C03636=1030.587,97.043,400.523,168.711,44.180,158.272
C03637=1030.581,96.794,400.543,168.708,44.181,158.272
C03638=1030.575,96.545,400.561,168.706,44.183,158.272
C03639=1030.569,96.295,400.580,168.703,44.185,158.272
C03640=1030.563,96.046,400.599,168.701,44.187,158.272
C03641=1030.556,95.797,400.618,168.699,44.189,158.273
C03642=1030.551,95.548,400.637,168.696,44.191,158.273
C03643=1030.544,95.298,400.656,168.694,44.193,158.273
C03644=1030.539,95.049,400.675,168.691,44.195,158.273
C03645=1030.532,94.800,400.694,168.689,44.197,158.273
C03646=1030.526,94.550,400.713,168.687,44.198,158.273
C03647=1030.520,94.301,400.731,168.684,44.200,158.273
C03648=1030.514,94.053,400.751,168.682,44.202,158.274
C03649=1030.508,93.803,400.770,168.679,44.204,158.274
C03650=1030.501,93.554,400.789,168.677,44.206,158.274
C03651=1030.496,93.305,400.808,168.675,44.208,158.274
C03652=1030.489,93.056,400.827,168.673,44.210,158.274
C03653=1030.483,92.806,400.846,168.670,44.211,158.274
C03654=1030.476,92.521,400.866,168.667,44.213,158.274
C03655=1030.469,92.236,400.888,168.665,44.215,158.275
C03656=1030.462,91.950,400.911,168.661,44.217,158.275
C03657=1030.455,91.665,400.932,168.659,44.219,158.275
C03658=1030.449,91.416,400.951,168.656,44.221,158.275
C03659=1030.443,91.166,400.970,168.654,44.223,158.275
C03660=1030.437,90.918,400.988,168.652,44.225,158.275
C03661=1030.431,90.669,401.007,168.649,44.227,158.275
C03662=1030.425,90.419,401.026,168.647,44.229,158.275
C03663=1030.419,90.170,401.045,168.644,44.231,158.276
C03664=1030.413,89.921,401.064,168.642,44.232,158.276
C03665=1030.407,89.672,401.083,168.640,44.234,158.276
C03666=1030.400,89.422,401.101,168.637,44.236,158.276
C03667=1030.394,89.173,401.119,168.635,44.238,158.276
C03668=1030.388,88.923,401.138,168.632,44.240,158.276
C03669=1030.382,88.674,401.157,168.631,44.242,158.277
C03670=1030.376,88.425,401.176,168.628,44.244,158.277
C03671=1030.369,88.176,401.194,168.625,44.245,158.277
C03672=1030.363,87.926,401.212,168.623,44.247,158.277
C03673=1030.357,87.677,401.231,168.620,44.249,158.277
C03674=1030.351,87.429,401.249,168.618,44.252,158.277
C03675=1030.345,87.179,401.269,168.616,44.254,158.278
C03676=1030.339,86.929,401.286,168.614,44.256,158.278
C03677=1030.333,86.680,401.305,168.611,44.257,158.278
C03678=1030.326,86.431,401.324,168.608,44.259,158.278
C03679=1030.320,86.182,401.342,168.606,44.261,158.278
C03680=1030.314,85.932,401.360,168.604,44.263,158.278
C03681=1030.307,85.683,401.379,168.602,44.265,158.278
C03682=1030.301,85.434,401.398,168.599,44.267,158.279
C03683=1030.296,85.185,401.417,168.597,44.269,158.279
C03684=1030.290,84.936,401.434,168.594,44.271,158.279
C03685=1030.283,84.686,401.453,168.591,44.273,158.279
C03686=1030.277,84.437,401.472,168.590,44.274,158.279
C03687=1030.271,84.188,401.490,168.587,44.276,158.279
C03688=1030.264,83.938,401.508,168.585,44.278,158.279
C03689=1030.258,83.689,401.527,168.582,44.280,158.280
C03690=1030.252,83.441,401.545,168.579,44.282,158.280
C03691=1030.246,83.191,401.563,168.578,44.284,158.280
C03692=1030.240,82.942,401.582,168.575,44.286,158.280
C03693=1030.234,82.693,401.601,168.573,44.288,158.280
C03694=1030.228,82.443,401.619,168.570,44.290,158.280
C03695=1030.222,82.194,401.637,168.567,44.291,158.280
C03696=1030.216,81.945,401.655,168.566,44.293,158.281
C03697=1030.209,81.696,401.674,168.563,44.295,158.281
C03698=1030.203,81.446,401.693,168.561,44.297,158.281
C03699=1030.197,81.197,401.710,168.558,44.299,158.281
C03700=1030.191,80.948,401.729,168.557,44.301,158.281
C03701=1030.185,80.698,401.747,168.554,44.303,158.281
C03702=1030.179,80.449,401.766,168.551,44.304,158.281
C03703=1030.173,80.200,401.785,168.549,44.306,158.282
C03704=1030.166,79.950,401.803,168.546,44.308,158.282
C03705=1030.161,79.702,401.821,168.545,44.310,158.282
C03706=1030.155,79.452,401.839,168.542,44.312,158.282
C03707=1030.148,79.203,401.857,168.539,44.314,158.282
C03708=1030.142,78.953,401.875,168.537,44.316,158.282
C03709=1030.136,78.705,401.894,168.535,44.318,158.282
C03710=1030.130,78.456,401.912,168.533,44.319,158.283
C03711=1030.124,78.206,401.930,168.530,44.321,158.283
C03712=1030.118,77.957,401.949,168.528,44.323,158.283
C03713=1030.112,77.708,401.967,168.525,44.325,158.283
C03714=1030.106,77.458,401.984,168.523,44.327,158.283
C03715=1030.099,77.209,402.003,168.521,44.329,158.283
C03716=1030.093,76.959,402.021,168.518,44.331,158.283
C03717=1030.087,76.711,402.039,168.516,44.333,158.284
C03718=1030.080,76.425,402.060,168.513,44.335,158.284
C03719=1030.073,76.140,402.081,168.511,44.337,158.284
C03720=1030.066,75.855,402.102,168.508,44.339,158.284
C03721=1030.059,75.569,402.122,168.505,44.342,158.284
C03722=1030.053,75.320,402.140,168.503,44.344,158.284
C03723=1030.046,75.070,402.158,168.501,44.346,158.285
C03724=1030.040,74.821,402.175,168.498,44.348,158.285
C03725=1030.034,74.572,402.194,168.495,44.349,158.285
C03726=1030.028,74.322,402.212,168.493,44.351,158.285
C03727=1030.022,74.073,402.229,168.490,44.353,158.285
C03728=1030.016,73.824,402.248,168.489,44.355,158.285
C03729=1030.009,73.575,402.265,168.486,44.357,158.285
C03730=1030.003,73.325,402.283,168.483,44.359,158.286
C03731=1029.997,73.076,402.302,168.481,44.361,158.286
C03732=1029.991,72.827,402.320,168.478,44.363,158.286
C03733=1029.985,72.577,402.338,168.477,44.365,158.286
C03734=1029.978,72.329,402.355,168.474,44.366,158.286
C03735=1029.972,72.079,402.373,168.471,44.368,158.286
C03736=1029.966,71.829,402.391,168.469,44.370,158.286
C03737=1029.960,71.580,402.409,168.466,44.372,158.287
C03738=1029.954,71.331,402.427,168.465,44.374,158.287
C03739=1029.947,71.082,402.445,168.462,44.376,158.287
C03740=1029.942,70.833,402.462,168.460,44.378,158.287
C03741=1029.936,70.583,402.480,168.457,44.380,158.287
C03742=1029.929,70.334,402.499,168.456,44.382,158.287
C03743=1029.924,70.085,402.516,168.453,44.384,158.288
C03744=1029.917,69.835,402.534,168.450,44.386,158.288
C03745=1029.911,69.586,402.552,168.448,44.388,158.288
C03746=1029.905,69.337,402.569,168.445,44.390,158.288
C03747=1029.899,69.087,402.588,168.444,44.392,158.288
C03748=1029.892,68.838,402.605,168.441,44.394,158.288
C03749=1029.886,68.589,402.623,168.439,44.395,158.288
C03750=1029.880,68.339,402.641,168.436,44.397,158.289
C03751=1029.874,68.091,402.658,168.433,44.399,158.289
C03752=1029.868,67.841,402.676,168.432,44.401,158.289
C03753=1029.862,67.591,402.694,168.429,44.403,158.289
C03754=1029.855,67.343,402.711,168.427,44.405,158.289
C03755=1029.849,67.093,402.729,168.424,44.407,158.289
C03756=1029.842,66.844,402.746,168.421,44.409,158.289
C03757=1029.837,66.595,402.764,168.419,44.411,158.290
C03758=1029.831,66.345,402.782,168.418,44.413,158.290
C03759=1029.824,66.096,402.799,168.415,44.415,158.290
C03760=1029.818,65.847,402.817,168.412,44.417,158.290
C03761=1029.811,65.597,402.834,168.410,44.419,158.290
C03762=1029.806,65.348,402.852,168.407,44.421,158.290
C03763=1029.800,65.098,402.870,168.406,44.423,158.290
C03764=1029.793,64.850,402.887,168.403,44.424,158.291
C03765=1029.787,64.600,402.905,168.400,44.426,158.291
C03766=1029.781,64.351,402.922,168.398,44.428,158.291
C03767=1029.775,64.101,402.940,168.395,44.430,158.291
C03768=1029.768,63.852,402.957,168.394,44.432,158.291
C03769=1029.763,63.603,402.974,168.391,44.434,158.291
C03770=1029.756,63.353,402.992,168.389,44.437,158.292
C03771=1029.750,63.104,403.009,168.386,44.439,158.292
C03772=1029.743,62.855,403.027,168.384,44.440,158.292
C03773=1029.736,62.606,403.044,168.381,44.442,158.292
C03774=1029.731,62.356,403.061,168.379,44.445,158.292
C03775=1029.724,62.106,403.078,168.377,44.447,158.292
C03776=1029.718,61.858,403.095,168.374,44.449,158.293
C03777=1029.712,61.608,403.113,168.372,44.451,158.293
C03778=1029.706,61.359,403.130,168.369,44.453,158.293
C03779=1029.699,61.110,403.147,168.367,44.455,158.293
C03780=1029.692,60.860,403.164,168.364,44.457,158.293
C03781=1029.687,60.611,403.182,168.362,44.459,158.293
C03782=1029.679,60.325,403.201,168.359,44.462,158.294
C03783=1029.672,60.040,403.222,168.357,44.464,158.294
C03784=1029.665,59.755,403.241,168.354,44.466,158.294
C03785=1029.658,59.469,403.261,168.351,44.468,158.294
C03786=1029.651,59.220,403.278,168.348,44.470,158.294
C03787=1029.645,58.970,403.294,168.347,44.472,158.294
C03788=1029.639,58.720,403.312,168.344,44.475,158.295
C03789=1029.633,58.472,403.329,168.342,44.477,158.295
C03790=1029.626,58.222,403.346,168.339,44.478,158.295
C03791=1029.620,57.973,403.363,168.337,44.480,158.295
C03792=1029.614,57.723,403.381,168.334,44.482,158.295
C03793=1029.607,57.475,403.398,168.332,44.484,158.295
C03794=1029.601,57.225,403.415,168.330,44.487,158.296
C03795=1029.595,56.975,403.432,168.328,44.489,158.296
C03796=1029.588,56.726,403.449,168.325,44.491,158.296
C03797=1029.582,56.477,403.466,168.322,44.492,158.296
C03798=1029.576,56.227,403.483,168.320,44.494,158.296
C03799=1029.570,55.978,403.500,168.318,44.496,158.296
C03800=1029.563,55.729,403.518,168.316,44.498,158.296
C03801=1029.557,55.479,403.534,168.313,44.501,158.297
C03802=1029.550,55.230,403.551,168.311,44.503,158.297
C03803=1029.545,54.981,403.569,168.308,44.505,158.297
C03804=1029.538,54.731,403.585,168.305,44.507,158.297
C03805=1029.532,54.482,403.602,168.303,44.508,158.297
C03806=1029.526,54.233,403.619,168.301,44.510,158.297
C03807=1029.520,53.983,403.637,168.299,44.512,158.297
C03808=1029.514,53.734,403.654,168.296,44.514,158.298
C03809=1029.507,53.485,403.671,168.294,44.517,158.298
C03810=1029.502,53.235,403.688,168.291,44.519,158.298
C03811=1029.495,52.986,403.705,168.290,44.520,158.298
C03812=1029.489,52.736,403.721,168.287,44.522,158.298
C03813=1029.483,52.488,403.738,168.284,44.524,158.298
C03814=1029.477,52.238,403.756,168.282,44.526,158.299
C03815=1029.471,51.989,403.772,168.279,44.528,158.299
C03816=1029.464,51.739,403.790,168.277,44.530,158.299
C03817=1029.458,51.490,403.806,168.275,44.532,158.299
C03818=1029.452,51.241,403.823,168.273,44.534,158.299
C03819=1029.446,50.991,403.840,168.270,44.536,158.299
C03820=1029.439,50.742,403.857,168.268,44.538,158.300
C03821=1029.433,50.493,403.873,168.265,44.540,158.300
C03822=1029.427,50.243,403.891,168.262,44.542,158.300
C03823=1029.421,49.994,403.908,168.261,44.544,158.300
C03824=1029.415,49.744,403.925,168.258,44.546,158.300
C03825=1029.408,49.495,403.942,168.256,44.548,158.300
C03826=1029.402,49.246,403.958,168.253,44.550,158.300
C03827=1029.396,48.996,403.976,168.251,44.552,158.300
C03828=1029.390,48.747,403.992,168.249,44.554,158.301
C03829=1029.384,48.498,404.009,168.246,44.555,158.301
C03830=1029.377,48.248,404.026,168.244,44.557,158.301
C03831=1029.372,47.999,404.043,168.241,44.559,158.301
C03832=1029.366,47.750,404.060,168.239,44.561,158.301
C03833=1029.360,47.500,404.076,168.237,44.563,158.301
C03834=1029.353,47.251,404.093,168.235,44.565,158.301
C03835=1029.347,47.002,404.110,168.232,44.567,158.302
C03836=1029.342,46.753,404.127,168.229,44.569,158.302
C03837=1029.335,46.503,404.144,168.227,44.571,158.302
C03838=1029.329,46.254,404.161,168.225,44.573,158.302
C03839=1029.323,46.005,404.177,168.223,44.575,158.302
C03840=1029.317,45.754,404.194,168.220,44.576,158.302
C03841=1029.311,45.505,404.211,168.217,44.578,158.302
C03842=1029.305,45.256,404.228,168.215,44.580,158.302
C03843=1029.299,45.007,404.245,168.213,44.582,158.303
C03844=1029.292,44.757,404.261,168.211,44.584,158.303
C03845=1029.287,44.508,404.278,168.208,44.586,158.303
C03846=1029.279,44.222,404.297,168.206,44.588,158.303
C03847=1029.273,43.936,404.316,168.203,44.591,158.303
C03848=1029.265,43.651,404.336,168.200,44.593,158.303
C03849=1029.259,43.365,404.354,168.197,44.595,158.303
C03850=1029.253,43.115,404.372,168.194,44.597,158.304
C03851=1029.247,42.866,404.388,168.193,44.598,158.304
C03852=1029.241,42.617,404.404,168.190,44.600,158.304
C03853=1029.235,42.367,404.421,168.188,44.602,158.304
C03854=1029.228,42.118,404.438,168.185,44.604,158.304
C03855=1029.222,41.868,404.454,168.183,44.606,158.304
C03856=1029.216,41.619,404.470,168.180,44.609,158.304
C03857=1029.210,41.370,404.487,168.178,44.611,158.305
C03858=1029.203,41.120,404.503,168.176,44.613,158.305
C03859=1029.197,40.871,404.520,168.173,44.614,158.305
C03860=1029.191,40.622,404.537,168.171,44.616,158.305
C03861=1029.185,40.372,404.553,168.168,44.618,158.305
C03862=1029.179,40.122,404.569,168.166,44.620,158.305
C03863=1029.172,39.873,404.585,168.163,44.622,158.305
C03864=1029.166,39.625,404.602,168.162,44.624,158.306
C03865=1029.160,39.375,404.618,168.159,44.626,158.306
C03866=1029.154,39.126,404.635,168.156,44.628,158.306
C03867=1029.147,38.876,404.651,168.154,44.630,158.306
C03868=1029.141,38.626,404.667,168.151,44.633,158.306
C03869=1029.135,38.377,404.684,168.149,44.634,158.306
C03870=1029.129,38.128,404.700,168.147,44.636,158.306
C03871=1029.124,37.878,404.716,168.145,44.638,158.307
C03872=1029.117,37.629,404.734,168.142,44.640,158.307
C03873=1029.111,37.380,404.750,168.140,44.642,158.307
C03874=1029.105,37.130,404.766,168.137,44.644,158.307
C03875=1029.098,36.881,404.782,168.134,44.646,158.307
C03876=1029.092,36.632,404.798,168.132,44.648,158.307
C03877=1029.086,36.382,404.815,168.130,44.650,158.307
C03878=1029.080,36.132,404.831,168.128,44.652,158.308
C03879=1029.073,35.883,404.846,168.125,44.654,158.308
C03880=1029.067,35.634,404.863,168.123,44.656,158.308
C03881=1029.061,35.385,404.879,168.120,44.658,158.308
C03882=1029.054,35.136,404.895,168.118,44.660,158.308
C03883=1029.048,34.886,404.911,168.115,44.662,158.308
C03884=1029.042,34.636,404.927,168.112,44.664,158.308
C03885=1029.036,34.386,404.943,168.110,44.667,158.309
C03886=1029.029,34.137,404.959,168.108,44.668,158.309
C03887=1029.024,33.888,404.975,168.106,44.670,158.309
C03888=1029.018,33.639,404.991,168.103,44.672,158.309
C03889=1029.010,33.389,405.007,168.101,44.674,158.309
C03890=1029.004,33.139,405.024,168.098,44.676,158.309
C03891=1028.998,32.890,405.040,168.096,44.678,158.309
C03892=1028.992,32.641,405.055,168.093,44.681,158.310
C03893=1028.986,32.392,405.072,168.091,44.683,158.310
C03894=1028.980,32.142,405.088,168.088,44.685,158.310
C03895=1028.973,31.893,405.103,168.086,44.687,158.310
C03896=1028.967,31.643,405.119,168.084,44.688,158.310
C03897=1028.962,31.394,405.135,168.081,44.690,158.310
C03898=1028.954,31.144,405.151,168.079,44.692,158.310
C03899=1028.948,30.895,405.168,168.076,44.694,158.311
C03900=1028.942,30.646,405.184,168.074,44.696,158.311
C03901=1028.936,30.397,405.200,168.071,44.699,158.311
C03902=1028.930,30.147,405.215,168.069,44.701,158.311
C03903=1028.924,29.897,405.231,168.067,44.703,158.311
C03904=1028.917,29.648,405.247,168.065,44.705,158.311
C03905=1028.911,29.399,405.263,168.062,44.707,158.311
C03906=1028.905,29.150,405.280,168.059,44.709,158.312
C03907=1028.899,28.900,405.295,168.057,44.710,158.312
C03908=1028.893,28.651,405.311,168.054,44.712,158.312
C03909=1028.887,28.401,405.327,168.052,44.714,158.312
C03910=1028.879,28.069,405.348,168.049,44.717,158.312
C03911=1028.870,27.738,405.369,168.046,44.720,158.312
C03912=1028.862,27.407,405.390,168.043,44.723,158.313
C03913=1028.854,27.075,405.411,168.039,44.726,158.313
C03914=1028.848,26.825,405.427,168.037,44.728,158.313
C03915=1028.841,26.576,405.442,168.034,44.729,158.313
C03916=1028.835,26.326,405.458,168.031,44.731,158.313
C03917=1028.829,26.077,405.474,168.029,44.733,158.313
C03918=1028.823,25.827,405.490,168.026,44.735,158.313
C03919=1028.816,25.578,405.505,168.024,44.737,158.314
C03920=1028.810,25.329,405.521,168.022,44.740,158.314
C03921=1028.804,25.079,405.537,168.020,44.742,158.314
C03922=1028.797,24.830,405.552,168.017,44.744,158.314
C03923=1028.792,24.580,405.568,168.015,44.746,158.314
C03924=1028.785,24.331,405.583,168.012,44.748,158.314
C03925=1028.779,24.082,405.600,168.009,44.750,158.314
C03926=1028.773,23.855,405.613,168.007,44.752,158.315
C03927=1028.767,23.628,405.627,168.005,44.753,158.315
C03928=1028.762,23.402,405.642,168.003,44.755,158.315
C03929=1028.756,23.175,405.656,168.000,44.757,158.315
C03930=1028.751,22.948,405.670,167.999,44.759,158.315
C03931=1028.745,22.723,405.684,167.996,44.761,158.315
C03932=1028.739,22.495,405.698,167.993,44.763,158.315
C03933=1028.734,22.269,405.712,167.992,44.765,158.316
C03934=1028.727,22.020,405.728,167.989,44.767,158.316
C03935=1028.721,21.770,405.744,167.987,44.769,158.316
C03936=1028.715,21.521,405.759,167.984,44.771,158.316
C03937=1028.709,21.271,405.775,167.982,44.773,158.316
C03938=1028.702,21.022,405.791,167.979,44.775,158.316
C03939=1028.696,20.772,405.805,167.977,44.777,158.316
C03940=1028.690,20.523,405.822,167.974,44.779,158.316
C03941=1028.684,20.273,405.837,167.971,44.781,158.317
C03942=1028.678,20.023,405.852,167.970,44.783,158.317
C03943=1028.672,19.775,405.868,167.967,44.785,158.317
C03944=1028.666,19.525,405.883,167.965,44.787,158.317
C03945=1028.660,19.276,405.899,167.962,44.789,158.317
C03946=1028.653,19.026,405.914,167.960,44.791,158.317
C03947=1028.646,18.777,405.929,167.957,44.793,158.317
C03948=1028.641,18.527,405.945,167.955,44.795,158.318
C03949=1028.634,18.277,405.960,167.952,44.797,158.318
C03950=1028.628,18.028,405.975,167.949,44.799,158.318
C03951=1028.621,17.779,405.990,167.947,44.801,158.318
C03952=1028.616,17.529,406.006,167.944,44.803,158.318
C03953=1028.609,17.280,406.022,167.942,44.806,158.318
C03954=1028.603,17.030,406.037,167.939,44.808,158.318
C03955=1028.598,16.781,406.052,167.937,44.810,158.319
C03956=1028.591,16.532,406.067,167.934,44.812,158.319
C03957=1028.585,16.282,406.082,167.932,44.814,158.319
C03958=1028.578,16.032,406.097,167.929,44.816,158.319
C03959=1028.572,15.783,406.114,167.928,44.817,158.319
C03960=1028.566,15.533,406.128,167.925,44.820,158.319
C03961=1028.559,15.284,406.143,167.923,44.822,158.319
C03962=1028.553,15.036,406.159,167.920,44.824,158.320
C03963=1028.548,14.786,406.174,167.917,44.826,158.320
C03964=1028.541,14.536,406.189,167.915,44.828,158.320
C03965=1028.535,14.286,406.204,167.912,44.830,158.320
C03966=1028.528,14.037,406.220,167.910,44.832,158.320
C03967=1028.523,13.787,406.235,167.907,44.834,158.320
C03968=1028.516,13.538,406.250,167.905,44.837,158.320
C03969=1028.510,13.289,406.265,167.902,44.839,158.320
C03970=1028.504,13.039,406.280,167.900,44.840,158.321
C03971=1028.498,12.789,406.295,167.897,44.842,158.321
C03972=1028.491,12.540,406.310,167.895,44.845,158.321
C03973=1028.485,12.291,406.325,167.892,44.847,158.321
C03974=1028.477,12.006,406.341,167.890,44.849,158.321
C03975=1028.470,11.721,406.359,167.886,44.852,158.321
C03976=1028.463,11.437,406.376,167.884,44.855,158.322
C03977=1028.456,11.153,406.393,167.880,44.857,158.322
C03978=1028.449,10.903,406.408,167.878,44.859,158.322
C03979=1028.443,10.653,406.423,167.875,44.861,158.322
C03980=1028.436,10.404,406.438,167.873,44.863,158.322
C03981=1028.430,10.154,406.453,167.870,44.865,158.322
C03982=1028.424,9.905,406.467,167.868,44.867,158.322
C03983=1028.418,9.655,406.482,167.865,44.869,158.323
C03984=1028.412,9.406,406.497,167.863,44.872,158.323
C03985=1028.405,9.156,406.512,167.860,44.874,158.323
C03986=1028.399,8.907,406.527,167.858,44.876,158.323
C03987=1028.393,8.657,406.541,167.855,44.878,158.323
C03988=1028.387,8.408,406.556,167.852,44.880,158.323
C03989=1028.380,8.158,406.571,167.850,44.882,158.323
C03990=1028.374,7.909,406.586,167.847,44.884,158.324
C03991=1028.368,7.659,406.601,167.845,44.886,158.324
C03992=1028.362,7.410,406.616,167.842,44.888,158.324
C03993=1028.355,7.160,406.631,167.840,44.890,158.324
C03994=1028.350,6.911,406.645,167.837,44.893,158.324
C03995=1028.343,6.662,406.660,167.835,44.895,158.324
C03996=1028.337,6.412,406.675,167.832,44.897,158.324
C03997=1028.330,6.162,406.690,167.830,44.899,158.325
C03998=1028.325,5.913,406.705,167.827,44.901,158.325
C03999=1028.318,5.664,406.720,167.824,44.903,158.325
C04000=1028.312,5.414,406.735,167.822,44.906,158.325
C04001=1028.306,5.165,406.749,167.820,44.908,158.325
C04002=1028.300,4.915,406.764,167.817,44.910,158.325
C04003=1028.293,4.666,406.779,167.814,44.912,158.325
C04004=1028.287,4.416,406.794,167.812,44.914,158.325
C04005=1028.281,4.166,406.808,167.809,44.915,158.326
C04006=1028.275,3.917,406.823,167.807,44.918,158.326
C04007=1028.269,3.667,406.838,167.804,44.920,158.326
C04008=1028.263,3.418,406.852,167.802,44.922,158.326
C04009=1028.256,3.169,406.867,167.799,44.924,158.326
C04010=1028.249,2.919,406.882,167.797,44.926,158.326
C04011=1028.244,2.670,406.896,167.794,44.928,158.326
C04012=1028.238,2.420,406.911,167.791,44.930,158.326
C04013=1028.232,2.171,406.925,167.789,44.932,158.327
C04014=1028.225,1.921,406.940,167.787,44.935,158.327
C04015=1028.219,1.672,406.955,167.784,44.937,158.327
C04016=1028.213,1.423,406.970,167.781,44.939,158.327
C04017=1028.207,1.172,406.984,167.779,44.941,158.327
C04018=1028.201,0.923,406.999,167.776,44.943,158.327
C04019=1028.195,0.674,407.013,167.774,44.945,158.327
C04020=1028.189,0.424,407.028,167.771,44.947,158.327
C04021=1028.183,0.175,407.043,167.768,44.949,158.328
C04022=1028.177,-0.075,407.057,167.766,44.951,158.328
C04023=1028.170,-0.325,407.072,167.763,44.952,158.328
C04024=1028.165,-0.574,407.087,167.761,44.954,158.328
C04025=1028.157,-0.823,407.101,167.758,44.957,158.328
C04026=1028.152,-1.073,407.115,167.756,44.959,158.328
C04027=1028.146,-1.322,407.130,167.753,44.961,158.328
C04028=1028.140,-1.571,407.144,167.751,44.963,158.328
C04029=1028.134,-1.821,407.159,167.748,44.965,158.329
C04030=1028.127,-2.071,407.174,167.746,44.967,158.329
C04031=1028.122,-2.320,407.188,167.743,44.969,158.329
C04032=1028.115,-2.570,407.203,167.740,44.971,158.329
C04033=1028.110,-2.819,407.217,167.738,44.973,158.329
C04034=1028.103,-3.069,407.232,167.735,44.975,158.329
C04035=1028.098,-3.318,407.246,167.733,44.977,158.329
C04036=1028.091,-3.568,407.261,167.730,44.979,158.329
C04037=1028.086,-3.817,407.275,167.727,44.981,158.329
C04038=1028.078,-4.100,407.291,167.725,44.984,158.330
C04039=1028.071,-4.382,407.308,167.722,44.986,158.330
C04040=1028.064,-4.665,407.323,167.719,44.988,158.330
C04041=1028.057,-4.948,407.339,167.716,44.991,158.330
C04042=1028.050,-5.197,407.353,167.713,44.993,158.330
C04043=1028.044,-5.447,407.368,167.711,44.995,158.330
C04044=1028.038,-5.696,407.382,167.708,44.997,158.331
C04045=1028.032,-5.946,407.396,167.706,44.999,158.331
C04046=1028.026,-6.195,407.410,167.703,45.002,158.331
C04047=1028.019,-6.445,407.424,167.701,45.004,158.331
C04048=1028.013,-6.694,407.439,167.698,45.006,158.331
C04049=1028.006,-6.944,407.452,167.696,45.008,158.331
C04050=1028.001,-7.194,407.466,167.693,45.010,158.331
C04051=1027.995,-7.443,407.481,167.691,45.013,158.332
C04052=1027.988,-7.693,407.494,167.688,45.015,158.332
C04053=1027.982,-7.942,407.509,167.684,45.017,158.332
C04054=1027.976,-8.191,407.523,167.682,45.019,158.332
C04055=1027.969,-8.441,407.538,167.680,45.021,158.332
C04056=1027.963,-8.690,407.551,167.677,45.023,158.332
C04057=1027.957,-8.941,407.565,167.674,45.025,158.332
C04058=1027.951,-9.190,407.580,167.672,45.027,158.332
C04059=1027.944,-9.440,407.593,167.669,45.029,158.332
C04060=1027.939,-9.689,407.607,167.667,45.032,158.333
C04061=1027.932,-9.938,407.622,167.664,45.034,158.333
C04062=1027.926,-10.188,407.635,167.662,45.036,158.333
C04063=1027.920,-10.437,407.649,167.659,45.038,158.333
C04064=1027.914,-10.687,407.664,167.657,45.040,158.333
C04065=1027.908,-10.936,407.677,167.653,45.042,158.333
C04066=1027.901,-11.186,407.692,167.651,45.045,158.333
C04067=1027.896,-11.435,407.706,167.648,45.047,158.334
C04068=1027.889,-11.685,407.719,167.645,45.049,158.334
C04069=1027.883,-11.935,407.733,167.643,45.051,158.334
C04070=1027.877,-12.184,407.747,167.640,45.053,158.334
C04071=1027.871,-12.434,407.761,167.638,45.055,158.334
C04072=1027.865,-12.683,407.775,167.635,45.057,158.334
C04073=1027.858,-12.933,407.790,167.633,45.059,158.334
C04074=1027.852,-13.182,407.803,167.630,45.061,158.334
C04075=1027.846,-13.432,407.817,167.628,45.063,158.335
C04076=1027.840,-13.682,407.830,167.625,45.065,158.335
C04077=1027.834,-13.931,407.845,167.622,45.068,158.335
C04078=1027.828,-14.180,407.859,167.619,45.070,158.335
C04079=1027.822,-14.430,407.872,167.617,45.072,158.335
C04080=1027.816,-14.680,407.886,167.614,45.074,158.335
C04081=1027.809,-14.930,407.900,167.611,45.076,158.335
C04082=1027.804,-15.179,407.915,167.609,45.078,158.335
C04083=1027.797,-15.428,407.928,167.606,45.080,158.335
C04084=1027.791,-15.678,407.942,167.604,45.082,158.336
C04085=1027.785,-15.927,407.955,167.601,45.085,158.336
C04086=1027.779,-16.177,407.969,167.599,45.087,158.336
C04087=1027.773,-16.427,407.983,167.595,45.089,158.336
C04088=1027.767,-16.676,407.996,167.593,45.091,158.336
C04089=1027.760,-16.926,408.009,167.590,45.094,158.336
C04090=1027.753,-17.176,408.023,167.588,45.096,158.336
C04091=1027.748,-17.425,408.037,167.585,45.098,158.337
C04092=1027.742,-17.674,408.050,167.583,45.100,158.337
C04093=1027.735,-17.924,408.064,167.579,45.103,158.337
C04094=1027.729,-18.173,408.078,167.577,45.105,158.337
C04095=1027.723,-18.423,408.092,167.574,45.107,158.337
C04096=1027.716,-18.672,408.105,167.572,45.109,158.337
C04097=1027.710,-18.922,408.118,167.569,45.111,158.337
C04098=1027.704,-19.171,408.132,167.567,45.113,158.337
C04099=1027.698,-19.421,408.146,167.564,45.115,158.338
C04100=1027.691,-19.671,408.159,167.560,45.118,158.338
C04101=1027.685,-19.920,408.173,167.558,45.120,158.338
C04102=1027.679,-20.202,408.188,167.556,45.122,158.338
C04103=1027.672,-20.483,408.203,167.552,45.125,158.338
C04104=1027.665,-20.763,408.218,167.550,45.127,158.338
C04105=1027.658,-21.044,408.233,167.546,45.130,158.338
C04106=1027.652,-21.294,408.246,167.544,45.132,158.339
C04107=1027.645,-21.544,408.260,167.541,45.134,158.339
C04108=1027.640,-21.793,408.274,167.539,45.136,158.339
C04109=1027.633,-22.043,408.287,167.535,45.139,158.339
C04110=1027.627,-22.292,408.300,167.533,45.141,158.339
C04111=1027.620,-22.542,408.314,167.530,45.143,158.339
C04112=1027.615,-22.791,408.328,167.527,45.145,158.339
C04113=1027.609,-23.041,408.340,167.525,45.147,158.339
C04114=1027.603,-23.290,408.354,167.523,45.150,158.340
C04115=1027.596,-23.540,408.367,167.519,45.152,158.340
C04116=1027.590,-23.790,408.381,167.516,45.154,158.340
C04117=1027.584,-24.039,408.394,167.514,45.156,158.340
C04118=1027.578,-24.289,408.408,167.511,45.158,158.340
C04119=1027.572,-24.538,408.421,167.509,45.161,158.340
C04120=1027.567,-24.788,408.434,167.506,45.163,158.340
C04121=1027.560,-25.038,408.448,167.504,45.165,158.340
C04122=1027.554,-25.287,408.461,167.500,45.167,158.340
C04123=1027.547,-25.537,408.474,167.498,45.169,158.340
C04124=1027.542,-25.786,408.488,167.495,45.171,158.341
C04125=1027.536,-26.036,408.501,167.493,45.173,158.341
C04126=1027.530,-26.285,408.514,167.490,45.175,158.341
C04127=1027.524,-26.534,408.527,167.488,45.177,158.341
C04128=1027.517,-26.785,408.542,167.484,45.180,158.341
C04129=1027.511,-27.034,408.555,167.481,45.182,158.341
C04130=1027.505,-27.284,408.567,167.479,45.184,158.341
C04131=1027.499,-27.533,408.581,167.476,45.186,158.342
C04132=1027.493,-27.782,408.594,167.474,45.188,158.342
C04133=1027.487,-28.032,408.606,167.470,45.191,158.342
C04134=1027.481,-28.282,408.620,167.468,45.193,158.342
C04135=1027.474,-28.532,408.633,167.465,45.195,158.342
C04136=1027.468,-28.781,408.646,167.463,45.197,158.342
C04137=1027.462,-29.031,408.659,167.461,45.200,158.342
C04138=1027.456,-29.281,408.672,167.457,45.202,158.342
C04139=1027.450,-29.530,408.685,167.454,45.204,158.342
C04140=1027.444,-29.780,408.698,167.452,45.207,158.343
C04141=1027.438,-30.029,408.711,167.449,45.209,158.343
C04142=1027.431,-30.278,408.724,167.446,45.211,158.343
C04143=1027.425,-30.529,408.737,167.443,45.213,158.343
C04144=1027.419,-30.778,408.750,167.441,45.216,158.343
C04145=1027.413,-31.028,408.763,167.438,45.218,158.343
C04146=1027.406,-31.277,408.776,167.436,45.220,158.343
C04147=1027.400,-31.527,408.788,167.432,45.223,158.344
C04148=1027.394,-31.776,408.801,167.430,45.225,158.344
C04149=1027.388,-32.026,408.814,167.427,45.227,158.344
C04150=1027.382,-32.275,408.827,167.425,45.229,158.344
C04151=1027.376,-32.525,408.840,167.421,45.232,158.344
C04152=1027.369,-32.774,408.853,167.419,45.234,158.344
C04153=1027.363,-33.024,408.866,167.416,45.236,158.344
C04154=1027.357,-33.274,408.879,167.414,45.238,158.344
C04155=1027.351,-33.523,408.891,167.411,45.240,158.345
C04156=1027.345,-33.773,408.905,167.408,45.243,158.345
C04157=1027.339,-34.023,408.917,167.405,45.245,158.345
C04158=1027.333,-34.272,408.930,167.403,45.247,158.345
C04159=1027.327,-34.522,408.943,167.400,45.249,158.345
C04160=1027.321,-34.771,408.956,167.397,45.251,158.345
C04161=1027.315,-35.021,408.969,167.394,45.254,158.345
C04162=1027.309,-35.271,408.981,167.392,45.256,158.345
C04163=1027.303,-35.520,408.995,167.389,45.258,158.346
C04164=1027.296,-35.770,409.007,167.386,45.260,158.346
C04165=1027.290,-36.019,409.020,167.383,45.262,158.346
C04166=1027.283,-36.300,409.034,167.381,45.265,158.346
C04167=1027.276,-36.580,409.049,167.377,45.267,158.346
C04168=1027.270,-36.860,409.062,167.374,45.270,158.346
C04169=1027.263,-37.140,409.077,167.371,45.272,158.346
C04170=1027.257,-37.390,409.090,167.368,45.275,158.346
C04171=1027.251,-37.639,409.103,167.365,45.277,158.346
C04172=1027.245,-37.889,409.116,167.363,45.279,158.347
C04173=1027.239,-38.139,409.128,167.360,45.281,158.347
C04174=1027.233,-38.388,409.141,167.358,45.283,158.347
C04175=1027.227,-38.638,409.154,167.354,45.285,158.347
C04176=1027.221,-38.888,409.167,167.352,45.288,158.347
C04177=1027.214,-39.137,409.178,167.349,45.290,158.347
C04178=1027.208,-39.386,409.192,167.346,45.292,158.347
C04179=1027.202,-39.636,409.204,167.343,45.295,158.347
C04180=1027.197,-39.886,409.216,167.341,45.297,158.347
C04181=1027.190,-40.135,409.228,167.338,45.299,158.348
C04182=1027.184,-40.385,409.241,167.335,45.302,158.348
C04183=1027.178,-40.635,409.254,167.332,45.304,158.348
C04184=1027.172,-40.884,409.266,167.330,45.307,158.348
C04185=1027.166,-41.134,409.279,167.326,45.309,158.348
C04186=1027.160,-41.384,409.291,167.324,45.311,158.348
C04187=1027.153,-41.633,409.303,167.321,45.314,158.348
C04188=1027.147,-41.883,409.316,167.319,45.316,158.349
C04189=1027.140,-42.133,409.328,167.315,45.318,158.349
C04190=1027.135,-42.382,409.340,167.313,45.321,158.349
C04191=1027.129,-42.631,409.353,167.310,45.323,158.349
C04192=1027.122,-42.881,409.365,167.307,45.325,158.349
C04193=1027.116,-43.131,409.378,167.304,45.328,158.349
C04194=1027.111,-43.380,409.390,167.302,45.330,158.349
C04195=1027.104,-43.630,409.402,167.298,45.332,158.349
C04196=1027.098,-43.880,409.415,167.296,45.335,158.350
C04197=1027.093,-44.129,409.427,167.293,45.337,158.350
C04198=1027.086,-44.379,409.439,167.291,45.339,158.350
C04199=1027.080,-44.629,409.452,167.287,45.342,158.350
C04200=1027.074,-44.878,409.464,167.285,45.344,158.350
C04201=1027.068,-45.128,409.476,167.282,45.346,158.350
C04202=1027.062,-45.377,409.488,167.279,45.348,158.350
C04203=1027.056,-45.627,409.501,167.276,45.350,158.350
C04204=1027.050,-45.877,409.513,167.274,45.353,158.350
C04205=1027.044,-46.127,409.525,167.270,45.355,158.351
C04206=1027.037,-46.376,409.537,167.268,45.357,158.351
C04207=1027.032,-46.625,409.549,167.265,45.359,158.351
C04208=1027.026,-46.875,409.562,167.263,45.361,158.351
C04209=1027.019,-47.125,409.574,167.259,45.364,158.351
C04210=1027.013,-47.375,409.587,167.257,45.366,158.351
C04211=1027.008,-47.624,409.599,167.254,45.368,158.351
C04212=1027.001,-47.873,409.611,167.251,45.371,158.351
C04213=1026.995,-48.123,409.623,167.248,45.373,158.352
C04214=1026.989,-48.373,409.635,167.246,45.375,158.352
C04215=1026.984,-48.622,409.647,167.242,45.378,158.352
C04216=1026.978,-48.872,409.660,167.240,45.380,158.352
C04217=1026.971,-49.122,409.671,167.237,45.382,158.352
C04218=1026.965,-49.372,409.684,167.234,45.385,158.352
C04219=1026.960,-49.621,409.696,167.231,45.387,158.352
C04220=1026.953,-49.871,409.708,167.229,45.389,158.352
C04221=1026.948,-50.121,409.720,167.226,45.391,158.352
C04222=1026.941,-50.369,409.732,167.223,45.394,158.352
C04223=1026.936,-50.619,409.745,167.220,45.396,158.353
C04224=1026.929,-50.870,409.756,167.218,45.398,158.353
C04225=1026.923,-51.119,409.768,167.214,45.401,158.353
C04226=1026.917,-51.368,409.780,167.212,45.403,158.353
C04227=1026.911,-51.618,409.791,167.208,45.406,158.353
C04228=1026.904,-51.868,409.803,167.206,45.408,158.353
C04229=1026.898,-52.118,409.816,167.203,45.411,158.354
C04230=1026.892,-52.398,409.828,167.200,45.413,158.354
C04231=1026.884,-52.679,409.842,167.197,45.416,158.354
C04232=1026.878,-52.960,409.855,167.193,45.419,158.354
C04233=1026.871,-53.240,409.868,167.190,45.422,158.354
C04234=1026.864,-53.489,409.880,167.187,45.424,158.354
C04235=1026.858,-53.739,409.891,167.184,45.427,158.354
C04236=1026.853,-53.989,409.903,167.181,45.429,158.354
C04237=1026.846,-54.239,409.915,167.179,45.432,158.355
C04238=1026.840,-54.488,409.927,167.175,45.434,158.355
C04239=1026.834,-54.737,409.938,167.173,45.437,158.355
C04240=1026.828,-54.988,409.950,167.170,45.439,158.355
C04241=1026.821,-55.237,409.962,167.167,45.442,158.355
C04242=1026.816,-55.487,409.973,167.165,45.444,158.355
C04243=1026.809,-55.736,409.985,167.161,45.447,158.355
C04244=1026.803,-55.986,409.996,167.159,45.449,158.356
C04245=1026.797,-56.236,410.008,167.155,45.452,158.356
C04246=1026.791,-56.485,410.020,167.153,45.454,158.356
C04247=1026.785,-56.735,410.031,167.150,45.456,158.356
C04248=1026.778,-56.984,410.043,167.147,45.458,158.356
C04249=1026.773,-57.234,410.054,167.145,45.461,158.356
C04250=1026.767,-57.484,410.067,167.141,45.463,158.356
C04251=1026.760,-57.734,410.078,167.139,45.466,158.357
C04252=1026.754,-57.983,410.089,167.135,45.468,158.357
C04253=1026.748,-58.233,410.101,167.133,45.471,158.357
C04254=1026.743,-58.482,410.113,167.130,45.473,158.357
C04255=1026.736,-58.732,410.124,167.127,45.476,158.357
C04256=1026.731,-58.982,410.135,167.124,45.478,158.357
C04257=1026.724,-59.231,410.147,167.121,45.480,158.357
C04258=1026.718,-59.482,410.158,167.118,45.483,158.357
C04259=1026.712,-59.731,410.170,167.116,45.485,158.357
C04260=1026.706,-59.981,410.182,167.112,45.488,158.358
C04261=1026.700,-60.230,410.193,167.110,45.490,158.358
C04262=1026.694,-60.480,410.204,167.107,45.493,158.358
C04263=1026.688,-60.730,410.215,167.104,45.495,158.358
C04264=1026.682,-60.979,410.228,167.101,45.498,158.358
C04265=1026.676,-61.229,410.239,167.098,45.500,158.358
C04266=1026.669,-61.478,410.251,167.096,45.503,158.358
C04267=1026.664,-61.728,410.262,167.092,45.505,158.358
C04268=1026.657,-61.978,410.273,167.090,45.507,158.359
C04269=1026.651,-62.227,410.284,167.086,45.510,158.359
C04270=1026.646,-62.478,410.296,167.084,45.512,158.359
C04271=1026.640,-62.727,410.307,167.081,45.515,158.359
C04272=1026.633,-62.977,410.319,167.078,45.517,158.359
C04273=1026.628,-63.226,410.330,167.075,45.520,158.359
C04274=1026.622,-63.476,410.341,167.072,45.522,158.359
C04275=1026.615,-63.725,410.353,167.069,45.524,158.359
C04276=1026.610,-63.975,410.364,167.067,45.527,158.360
C04277=1026.604,-64.225,410.375,167.063,45.529,158.360
C04278=1026.598,-64.475,410.386,167.061,45.532,158.360
C04279=1026.592,-64.724,410.398,167.058,45.534,158.360
C04280=1026.586,-64.974,410.409,167.055,45.536,158.360
C04281=1026.580,-65.223,410.420,167.052,45.539,158.360
C04282=1026.574,-65.474,410.432,167.049,45.541,158.360
C04283=1026.568,-65.723,410.443,167.047,45.544,158.360
C04284=1026.562,-65.973,410.455,167.043,45.546,158.360
C04285=1026.556,-66.222,410.466,167.041,45.548,158.361
C04286=1026.551,-66.472,410.476,167.037,45.551,158.361
C04287=1026.544,-66.721,410.488,167.035,45.553,158.361
C04288=1026.539,-66.971,410.500,167.032,45.556,158.361
C04289=1026.533,-67.221,410.511,167.029,45.558,158.361
C04290=1026.527,-67.471,410.522,167.026,45.560,158.361
C04291=1026.521,-67.720,410.533,167.023,45.563,158.361
C04292=1026.515,-67.970,410.544,167.020,45.565,158.361
C04293=1026.509,-68.219,410.556,167.017,45.568,158.362
C04294=1026.503,-68.501,410.568,167.014,45.570,158.362
C04295=1026.496,-68.783,410.580,167.011,45.573,158.362
C04296=1026.490,-69.065,410.593,167.008,45.576,158.362
C04297=1026.483,-69.346,410.606,167.004,45.578,158.362
C04298=1026.477,-69.596,410.618,167.002,45.581,158.362
C04299=1026.471,-69.846,410.629,166.998,45.583,158.362
C04300=1026.465,-70.095,410.639,166.996,45.585,158.362
C04301=1026.460,-70.345,410.650,166.992,45.588,158.362
C04302=1026.453,-70.595,410.661,166.990,45.590,158.363
C04303=1026.447,-70.845,410.672,166.987,45.592,158.363
C04304=1026.442,-71.094,410.684,166.984,45.595,158.363
C04305=1026.436,-71.345,410.695,166.981,45.597,158.363
C04306=1026.430,-71.594,410.706,166.978,45.599,158.363
C04307=1026.425,-71.844,410.717,166.975,45.602,158.363
C04308=1026.419,-72.093,410.728,166.973,45.604,158.363
C04309=1026.413,-72.343,410.739,166.969,45.607,158.363
C04310=1026.407,-72.593,410.750,166.967,45.609,158.363
C04311=1026.401,-72.842,410.761,166.963,45.611,158.363
C04312=1026.395,-73.092,410.772,166.961,45.614,158.364
C04313=1026.390,-73.342,410.783,166.957,45.616,158.364
C04314=1026.384,-73.592,410.794,166.955,45.618,158.364
C04315=1026.378,-73.841,410.805,166.952,45.621,158.364
C04316=1026.373,-74.091,410.816,166.949,45.623,158.364
C04317=1026.367,-74.340,410.827,166.946,45.626,158.364
C04318=1026.360,-74.590,410.838,166.943,45.628,158.364
C04319=1026.355,-74.840,410.849,166.940,45.631,158.364
C04320=1026.349,-75.089,410.860,166.937,45.633,158.365
C04321=1026.343,-75.339,410.870,166.935,45.636,158.365
C04322=1026.336,-75.589,410.881,166.931,45.638,158.365
C04323=1026.331,-75.839,410.892,166.929,45.641,158.365
C04324=1026.325,-76.088,410.903,166.925,45.643,158.365
C04325=1026.319,-76.338,410.913,166.923,45.646,158.365
C04326=1026.314,-76.588,410.924,166.919,45.648,158.365
C04327=1026.307,-76.837,410.934,166.917,45.651,158.365
C04328=1026.301,-77.087,410.945,166.913,45.653,158.365
C04329=1026.295,-77.337,410.956,166.911,45.656,158.366
C04330=1026.290,-77.586,410.967,166.908,45.658,158.366
C04331=1026.284,-77.836,410.977,166.905,45.661,158.366
C04332=1026.278,-78.086,410.987,166.902,45.663,158.366
C04333=1026.272,-78.335,410.998,166.899,45.666,158.366
C04334=1026.266,-78.586,411.009,166.896,45.668,158.366
C04335=1026.260,-78.835,411.020,166.893,45.671,158.366
C04336=1026.254,-79.085,411.030,166.890,45.673,158.366
C04337=1026.249,-79.334,411.041,166.888,45.676,158.367
C04338=1026.242,-79.584,411.051,166.884,45.678,158.367
C04339=1026.237,-79.834,411.062,166.882,45.681,158.367
C04340=1026.231,-80.084,411.072,166.879,45.683,158.367
C04341=1026.226,-80.333,411.083,166.876,45.686,158.367
C04342=1026.218,-80.583,411.093,166.872,45.689,158.367
C04343=1026.213,-80.833,411.104,166.870,45.691,158.367
C04344=1026.207,-81.082,411.114,166.867,45.694,158.368
C04345=1026.201,-81.333,411.124,166.864,45.697,158.368
C04346=1026.195,-81.582,411.134,166.861,45.699,158.368
C04347=1026.189,-81.832,411.144,166.858,45.702,158.368
C04348=1026.183,-82.081,411.155,166.855,45.705,158.368
C04349=1026.177,-82.331,411.165,166.851,45.707,158.368
C04350=1026.172,-82.581,411.176,166.849,45.710,158.368
C04351=1026.165,-82.830,411.185,166.846,45.713,158.369
C04352=1026.160,-83.080,411.196,166.843,45.715,158.369
C04353=1026.153,-83.330,411.206,166.840,45.718,158.369
C04354=1026.147,-83.580,411.217,166.838,45.721,158.369
C04355=1026.141,-83.830,411.227,166.834,45.723,158.369
C04356=1026.135,-84.079,411.238,166.832,45.726,158.369
C04357=1026.129,-84.329,411.247,166.828,45.729,158.369
C04358=1026.123,-84.613,411.259,166.825,45.732,158.370
C04359=1026.116,-84.896,411.270,166.822,45.735,158.370
C04360=1026.109,-85.180,411.282,166.818,45.738,158.370
C04361=1026.103,-85.464,411.294,166.815,45.741,158.370
C04362=1026.097,-85.714,411.303,166.811,45.743,158.370
C04363=1026.091,-85.964,411.314,166.809,45.746,158.370
C04364=1026.085,-86.214,411.324,166.806,45.749,158.370
C04365=1026.079,-86.463,411.335,166.803,45.751,158.370
C04366=1026.073,-86.713,411.344,166.800,45.754,158.371
C04367=1026.067,-86.963,411.354,166.796,45.757,158.371
C04368=1026.061,-87.212,411.365,166.794,45.759,158.371
C04369=1026.056,-87.462,411.375,166.791,45.762,158.371
C04370=1026.049,-87.712,411.384,166.788,45.764,158.371
C04371=1026.044,-87.961,411.395,166.785,45.767,158.371
C04372=1026.037,-88.211,411.405,166.782,45.769,158.371
C04373=1026.032,-88.461,411.415,166.779,45.772,158.372
C04374=1026.026,-88.711,411.425,166.776,45.774,158.372
C04375=1026.020,-88.961,411.436,166.773,45.777,158.372
C04376=1026.014,-89.210,411.445,166.770,45.780,158.372
C04377=1026.009,-89.460,411.455,166.767,45.782,158.372
C04378=1026.003,-89.709,411.465,166.764,45.785,158.372
C04379=1025.997,-89.959,411.475,166.761,45.787,158.372
C04380=1025.991,-90.209,411.485,166.758,45.790,158.372
C04381=1025.986,-90.459,411.495,166.756,45.793,158.373
C04382=1025.979,-90.708,411.505,166.752,45.795,158.373
C04383=1025.974,-90.958,411.515,166.750,45.798,158.373
C04384=1025.968,-91.208,411.525,166.746,45.800,158.373
C04385=1025.962,-91.458,411.535,166.743,45.803,158.373
C04386=1025.957,-91.707,411.544,166.741,45.806,158.373
C04387=1025.951,-91.957,411.555,166.737,45.808,158.373
C04388=1025.945,-92.207,411.565,166.735,45.811,158.373
C04389=1025.939,-92.457,411.575,166.731,45.813,158.373
C04390=1025.933,-92.707,411.585,166.729,45.816,158.374
C04391=1025.928,-92.957,411.595,166.725,45.819,158.374
C04392=1025.922,-93.206,411.604,166.723,45.821,158.374
C04393=1025.916,-93.455,411.615,166.720,45.824,158.374
C04394=1025.910,-93.705,411.624,166.716,45.827,158.374
C04395=1025.905,-93.955,411.635,166.714,45.829,158.374
C04396=1025.898,-94.205,411.644,166.710,45.832,158.374
C04397=1025.894,-94.454,411.654,166.708,45.834,158.374
C04398=1025.887,-94.704,411.663,166.704,45.837,158.375
C04399=1025.882,-94.954,411.674,166.702,45.840,158.375
C04400=1025.876,-95.204,411.683,166.699,45.842,158.375
C04401=1025.870,-95.454,411.693,166.696,45.845,158.375
C04402=1025.865,-95.703,411.703,166.693,45.847,158.375
C04403=1025.859,-95.953,411.713,166.690,45.850,158.375
C04404=1025.853,-96.203,411.723,166.687,45.852,158.375
C04405=1025.847,-96.452,411.733,166.683,45.855,158.375
C04406=1025.842,-96.702,411.742,166.681,45.858,158.376
C04407=1025.836,-96.952,411.752,166.678,45.860,158.376
C04408=1025.830,-97.202,411.762,166.675,45.863,158.376
C04409=1025.825,-97.451,411.771,166.672,45.866,158.376
C04410=1025.819,-97.701,411.781,166.669,45.868,158.376
C04411=1025.813,-97.951,411.791,166.666,45.871,158.376
C04412=1025.807,-98.201,411.800,166.663,45.874,158.376
C04413=1025.802,-98.450,411.809,166.660,45.876,158.376
C04414=1025.796,-98.700,411.819,166.657,45.879,158.377
C04415=1025.790,-98.950,411.829,166.654,45.882,158.377
C04416=1025.784,-99.200,411.838,166.651,45.885,158.377
C04417=1025.778,-99.449,411.848,166.648,45.887,158.377
C04418=1025.772,-99.699,411.857,166.645,45.890,158.377
C04419=1025.767,-99.950,411.867,166.642,45.893,158.377
C04420=1025.762,-100.199,411.876,166.639,45.896,158.377
C04421=1025.755,-100.448,411.885,166.636,45.898,158.378
C04422=1025.749,-100.735,411.896,166.633,45.902,158.378
C04423=1025.742,-101.020,411.907,166.630,45.905,158.378
C04424=1025.735,-101.307,411.918,166.625,45.908,158.378
C04425=1025.729,-101.592,411.928,166.622,45.911,158.378
C04426=1025.723,-101.843,411.938,166.620,45.914,158.378
C04427=1025.718,-102.092,411.948,166.616,45.917,158.379
C04428=1025.712,-102.342,411.956,166.613,45.919,158.379
C04429=1025.706,-102.592,411.966,166.610,45.922,158.379
C04430=1025.700,-102.841,411.975,166.607,45.925,158.379
C04431=1025.694,-103.091,411.985,166.605,45.928,158.379
C04432=1025.689,-103.342,411.994,166.601,45.930,158.379
C04433=1025.683,-103.591,412.003,166.598,45.933,158.379
C04434=1025.677,-103.840,412.013,166.596,45.936,158.380
C04435=1025.672,-104.090,412.021,166.592,45.939,158.380
C04436=1025.666,-104.340,412.031,166.590,45.941,158.380
C04437=1025.659,-104.590,412.041,166.586,45.944,158.380
C04438=1025.655,-104.840,412.050,166.583,45.947,158.380
C04439=1025.649,-105.090,412.059,166.581,45.950,158.380
C04440=1025.643,-105.339,412.068,166.577,45.952,158.380
C04441=1025.637,-105.589,412.077,166.574,45.955,158.380
C04442=1025.632,-105.838,412.087,166.572,45.958,158.381
C04443=1025.626,-106.088,412.096,166.568,45.961,158.381
C04444=1025.620,-106.338,412.105,166.566,45.963,158.381
C04445=1025.614,-106.587,412.114,166.562,45.966,158.381
C04446=1025.609,-106.838,412.124,166.559,45.969,158.381
C04447=1025.603,-107.087,412.133,166.557,45.971,158.381
C04448=1025.598,-107.338,412.142,166.553,45.974,158.381
C04449=1025.592,-107.587,412.151,166.550,45.977,158.381
C04450=1025.586,-107.837,412.160,166.547,45.979,158.382
C04451=1025.581,-108.086,412.169,166.544,45.982,158.382
C04452=1025.574,-108.336,412.178,166.542,45.985,158.382
C04453=1025.569,-108.586,412.187,166.538,45.988,158.382
C04454=1025.563,-108.836,412.197,166.535,45.991,158.382
C04455=1025.558,-109.085,412.205,166.533,45.993,158.382
C04456=1025.552,-109.336,412.214,166.529,45.996,158.382
C04457=1025.546,-109.585,412.223,166.526,45.999,158.383
C04458=1025.540,-109.835,412.232,166.524,46.002,158.383
C04459=1025.534,-110.084,412.241,166.520,46.005,158.383
C04460=1025.528,-110.334,412.249,166.517,46.008,158.383
C04461=1025.523,-110.584,412.259,166.515,46.011,158.383
C04462=1025.517,-110.834,412.267,166.511,46.013,158.383
C04463=1025.511,-111.084,412.276,166.508,46.016,158.383
C04464=1025.505,-111.334,412.285,166.505,46.019,158.384
C04465=1025.500,-111.583,412.294,166.502,46.022,158.384
C04466=1025.494,-111.832,412.303,166.499,46.025,158.384
C04467=1025.489,-112.083,412.312,166.497,46.028,158.384
C04468=1025.483,-112.332,412.320,166.493,46.030,158.384
C04469=1025.477,-112.582,412.330,166.490,46.033,158.384
C04470=1025.472,-112.832,412.339,166.487,46.036,158.385
C04471=1025.467,-113.082,412.347,166.484,46.039,158.385
C04472=1025.460,-113.331,412.357,166.481,46.042,158.385
C04473=1025.455,-113.581,412.365,166.478,46.045,158.385
C04474=1025.449,-113.832,412.374,166.475,46.047,158.385
C04475=1025.444,-114.081,412.383,166.472,46.050,158.385
C04476=1025.438,-114.330,412.392,166.469,46.053,158.385
C04477=1025.432,-114.581,412.400,166.466,46.056,158.385
C04478=1025.427,-114.830,412.408,166.464,46.059,158.386
C04479=1025.420,-115.080,412.418,166.460,46.062,158.386
C04480=1025.415,-115.330,412.426,166.457,46.065,158.386
C04481=1025.410,-115.579,412.435,166.455,46.067,158.386
C04482=1025.404,-115.830,412.444,166.451,46.070,158.386
C04483=1025.398,-116.079,412.452,166.448,46.073,158.386
C04484=1025.392,-116.328,412.461,166.445,46.075,158.387
C04485=1025.387,-116.579,412.470,166.442,46.078,158.387
C04486=1025.380,-116.864,412.480,166.439,46.082,158.387
C04487=1025.375,-117.150,412.489,166.435,46.085,158.387
C04488=1025.368,-117.436,412.499,166.431,46.088,158.387
C04489=1025.361,-117.721,412.509,166.428,46.092,158.387
C04490=1025.356,-117.971,412.517,166.425,46.095,158.388
C04491=1025.350,-118.222,412.526,166.422,46.097,158.388
C04492=1025.344,-118.471,412.534,166.419,46.100,158.388
C04493=1025.338,-118.721,412.543,166.416,46.103,158.388
C04494=1025.333,-118.970,412.551,166.413,46.106,158.388
C04495=1025.327,-119.221,412.560,166.410,46.109,158.388
C04496=1025.321,-119.470,412.568,166.407,46.112,158.388
C04497=1025.316,-119.720,412.576,166.404,46.115,158.389
C04498=1025.310,-119.970,412.586,166.401,46.118,158.389
C04499=1025.305,-120.219,412.594,166.398,46.121,158.389
C04500=1025.299,-120.469,412.602,166.396,46.124,158.389
C04501=1025.293,-120.719,412.611,166.392,46.127,158.389
C04502=1025.287,-120.969,412.620,166.389,46.130,158.389
C04503=1025.282,-121.219,412.628,166.387,46.132,158.390
C04504=1025.276,-121.468,412.636,166.383,46.135,158.390
C04505=1025.271,-121.718,412.644,166.380,46.138,158.390
C04506=1025.266,-121.967,412.653,166.378,46.141,158.390
C04507=1025.259,-122.218,412.661,166.374,46.144,158.390
C04508=1025.254,-122.467,412.670,166.371,46.147,158.390
C04509=1025.249,-122.718,412.677,166.368,46.149,158.390
C04510=1025.243,-122.967,412.685,166.365,46.152,158.390
C04511=1025.238,-123.217,412.694,166.362,46.155,158.391
C04512=1025.232,-123.467,412.703,166.360,46.158,158.391
C04513=1025.226,-123.717,412.711,166.356,46.161,158.391
C04514=1025.220,-123.966,412.719,166.353,46.164,158.391
C04515=1025.215,-124.216,412.727,166.351,46.167,158.391
C04516=1025.210,-124.466,412.736,166.347,46.170,158.391
C04517=1025.203,-124.716,412.744,166.344,46.173,158.392
C04518=1025.198,-124.966,412.752,166.341,46.176,158.392
C04519=1025.192,-125.216,412.760,166.338,46.179,158.392
C04520=1025.187,-125.465,412.768,166.335,46.182,158.392
C04521=1025.181,-125.715,412.776,166.332,46.185,158.392
C04522=1025.176,-125.964,412.785,166.329,46.188,158.392
C04523=1025.171,-126.215,412.793,166.326,46.191,158.393
C04524=1025.164,-126.465,412.801,166.323,46.194,158.393
C04525=1025.159,-126.715,412.809,166.320,46.197,158.393
C04526=1025.153,-126.964,412.817,166.317,46.200,158.393
C04527=1025.148,-127.214,412.826,166.314,46.203,158.393
C04528=1025.142,-127.464,412.833,166.310,46.206,158.393
C04529=1025.137,-127.713,412.841,166.308,46.208,158.393
C04530=1025.131,-127.963,412.849,166.305,46.212,158.394
C04531=1025.126,-128.213,412.858,166.303,46.214,158.394
C04532=1025.122,-128.462,412.866,166.299,46.217,158.394
C04533=1025.117,-128.712,412.877,166.296,46.218,158.394
C04534=1025.114,-128.962,412.888,166.294,46.218,158.394
C04535=1025.111,-129.211,412.898,166.291,46.219,158.393
C04536=1025.109,-129.461,412.910,166.289,46.220,158.393
C04537=1025.106,-129.710,412.922,166.287,46.219,158.393
C04538=1025.106,-129.961,412.934,166.284,46.218,158.392
C04539=1025.105,-130.210,412.947,166.281,46.217,158.392
C04540=1025.105,-130.460,412.961,166.279,46.215,158.391
C04541=1025.105,-130.709,412.976,166.278,46.213,158.391
C04542=1025.106,-130.960,412.990,166.275,46.210,158.390
C04543=1025.108,-131.209,413.006,166.274,46.207,158.389
C04544=1025.109,-131.459,413.023,166.271,46.203,158.388
C04545=1025.112,-131.709,413.039,166.270,46.199,158.387
C04546=1025.114,-131.959,413.057,166.268,46.194,158.387
C04547=1025.118,-132.209,413.074,166.267,46.188,158.385
C04548=1025.122,-132.458,413.093,166.265,46.183,158.384
C04549=1025.127,-132.708,413.112,166.264,46.177,158.383
C04550=1024.827,-132.734,412.781,166.216,46.449,158.423
C04551=1024.822,-132.484,412.763,166.218,46.456,158.425
C04552=1024.818,-132.235,412.744,166.219,46.462,158.426
C04553=1024.814,-131.985,412.726,166.221,46.467,158.427
C04554=1024.811,-131.734,412.708,166.221,46.471,158.428
C04555=1024.809,-131.485,412.692,166.224,46.476,158.429
C04556=1024.807,-131.236,412.676,166.226,46.479,158.429
C04557=1024.805,-130.986,412.660,166.227,46.483,158.430
C04558=1024.805,-130.735,412.645,166.229,46.485,158.431
C04559=1024.804,-130.486,412.630,166.231,46.488,158.432
C04560=1024.804,-130.236,412.617,166.234,46.490,158.432
C04561=1024.805,-129.986,412.604,166.236,46.491,158.433
C04562=1024.807,-129.737,412.591,166.238,46.492,158.433
C04563=1024.808,-129.487,412.579,166.241,46.492,158.433
C04564=1024.811,-129.236,412.568,166.243,46.492,158.433
C04565=1024.813,-128.987,412.557,166.246,46.491,158.434
C04566=1024.817,-128.737,412.546,166.249,46.490,158.434
C04567=1024.821,-128.488,412.537,166.252,46.489,158.434
C04568=1024.826,-128.238,412.528,166.254,46.487,158.434
C04569=1024.830,-127.988,412.518,166.257,46.484,158.434
C04570=1024.836,-127.739,412.511,166.260,46.481,158.434
C04571=1024.841,-127.489,412.502,166.263,46.478,158.434
C04572=1024.847,-127.240,412.494,166.266,46.475,158.433
C04573=1024.852,-126.989,412.486,166.269,46.472,158.433
C04574=1024.858,-126.740,412.479,166.272,46.469,158.433
C04575=1024.864,-126.490,412.470,166.275,46.466,158.433
C04576=1024.870,-126.241,412.462,166.278,46.463,158.433
C04577=1024.875,-125.991,412.454,166.281,46.460,158.433
C04578=1024.881,-125.741,412.447,166.284,46.457,158.433
C04579=1024.886,-125.491,412.438,166.287,46.453,158.432
C04580=1024.892,-125.241,412.429,166.290,46.450,158.432
C04581=1024.898,-124.992,412.421,166.293,46.447,158.432
C04582=1024.903,-124.741,412.414,166.296,46.444,158.432
C04583=1024.909,-124.492,412.406,166.300,46.441,158.432
C04584=1024.914,-124.242,412.397,166.302,46.438,158.431
C04585=1024.920,-123.992,412.388,166.305,46.435,158.431
C04586=1024.926,-123.742,412.380,166.308,46.432,158.431
C04587=1024.931,-123.493,412.372,166.311,46.429,158.431
C04588=1024.936,-123.242,412.364,166.314,46.426,158.431
C04589=1024.942,-122.993,412.356,166.317,46.423,158.431
C04590=1024.947,-122.743,412.348,166.321,46.420,158.431
C04591=1024.953,-122.493,412.339,166.323,46.418,158.430
C04592=1024.958,-122.243,412.330,166.326,46.414,158.430
C04593=1024.964,-121.994,412.323,166.330,46.411,158.430
C04594=1024.970,-121.744,412.314,166.332,46.409,158.430
C04595=1024.975,-121.494,412.306,166.335,46.406,158.430
C04596=1024.982,-121.244,412.297,166.338,46.403,158.430
C04597=1024.987,-120.994,412.289,166.342,46.399,158.430
C04598=1024.992,-120.745,412.280,166.344,46.397,158.429
C04599=1024.997,-120.495,412.272,166.347,46.394,158.429
C04600=1025.003,-120.246,412.264,166.351,46.391,158.429
C04601=1025.009,-119.995,412.255,166.353,46.388,158.429
C04602=1025.014,-119.745,412.247,166.356,46.385,158.429
C04603=1025.020,-119.496,412.238,166.360,46.382,158.429
C04604=1025.026,-119.246,412.230,166.363,46.379,158.428
C04605=1025.032,-118.996,412.221,166.365,46.376,158.428
C04606=1025.037,-118.746,412.213,166.368,46.373,158.428
C04607=1025.042,-118.496,412.204,166.372,46.370,158.428
C04608=1025.048,-118.247,412.197,166.374,46.367,158.428
C04609=1025.054,-117.997,412.188,166.377,46.364,158.428
C04610=1025.060,-117.748,412.178,166.381,46.361,158.428
C04611=1025.066,-117.461,412.169,166.384,46.358,158.427
C04612=1025.073,-117.176,412.159,166.387,46.354,158.427
C04613=1025.078,-116.891,412.149,166.391,46.351,158.427
C04614=1025.085,-116.605,412.139,166.395,46.348,158.427
C04615=1025.091,-116.355,412.131,166.397,46.345,158.427
C04616=1025.097,-116.105,412.123,166.400,46.342,158.427
C04617=1025.102,-115.855,412.114,166.404,46.339,158.426
C04618=1025.108,-115.606,412.106,166.407,46.336,158.426
C04619=1025.114,-115.355,412.097,166.409,46.333,158.426
C04620=1025.119,-115.106,412.088,166.412,46.330,158.426
C04621=1025.124,-114.856,412.079,166.416,46.327,158.426
C04622=1025.131,-114.606,412.071,166.418,46.324,158.426
C04623=1025.136,-114.357,412.062,166.421,46.321,158.426
C04624=1025.142,-114.107,412.053,166.425,46.318,158.425
C04625=1025.148,-113.857,412.044,166.428,46.315,158.425
C04626=1025.153,-113.607,412.036,166.430,46.312,158.425
C04627=1025.159,-113.357,412.027,166.434,46.309,158.425
C04628=1025.164,-113.108,412.018,166.437,46.306,158.425
C04629=1025.170,-112.858,412.009,166.439,46.304,158.425
C04630=1025.176,-112.608,412.000,166.443,46.301,158.425
C04631=1025.181,-112.359,411.991,166.446,46.298,158.424
C04632=1025.187,-112.108,411.982,166.448,46.295,158.424
C04633=1025.192,-111.859,411.974,166.452,46.292,158.424
C04634=1025.198,-111.609,411.965,166.455,46.289,158.424
C04635=1025.204,-111.359,411.956,166.457,46.286,158.424
C04636=1025.210,-111.110,411.948,166.461,46.283,158.424
C04637=1025.216,-110.860,411.938,166.464,46.280,158.423
C04638=1025.221,-110.610,411.930,166.466,46.278,158.423
C04639=1025.227,-110.360,411.920,166.469,46.275,158.423
C04640=1025.233,-110.111,411.912,166.473,46.272,158.423
C04641=1025.238,-109.860,411.903,166.475,46.269,158.423
C04642=1025.244,-109.611,411.894,166.479,46.266,158.423
C04643=1025.249,-109.361,411.885,166.482,46.263,158.423
C04644=1025.255,-109.112,411.876,166.485,46.260,158.423
C04645=1025.261,-108.862,411.867,166.487,46.258,158.422
C04646=1025.267,-108.612,411.858,166.491,46.255,158.422
C04647=1025.272,-108.362,411.849,166.494,46.252,158.422
C04648=1025.278,-108.112,411.840,166.496,46.249,158.422
C04649=1025.284,-107.863,411.831,166.500,46.246,158.422
C04650=1025.289,-107.612,411.822,166.503,46.243,158.422
C04651=1025.295,-107.363,411.813,166.505,46.240,158.421
C04652=1025.301,-107.114,411.804,166.509,46.238,158.421
C04653=1025.306,-106.864,411.795,166.512,46.235,158.421
C04654=1025.313,-106.614,411.785,166.514,46.232,158.421
C04655=1025.318,-106.364,411.777,166.518,46.229,158.421
C04656=1025.324,-106.115,411.767,166.521,46.226,158.421
C04657=1025.329,-105.864,411.758,166.523,46.223,158.421
C04658=1025.335,-105.615,411.749,166.527,46.221,158.421
C04659=1025.341,-105.365,411.739,166.530,46.218,158.420
C04660=1025.346,-105.115,411.731,166.533,46.215,158.420
C04661=1025.352,-104.865,411.721,166.536,46.212,158.420
C04662=1025.358,-104.616,411.712,166.539,46.209,158.420
C04663=1025.364,-104.366,411.703,166.541,46.206,158.420
C04664=1025.369,-104.116,411.693,166.545,46.204,158.420
C04665=1025.374,-103.866,411.684,166.548,46.201,158.420
C04666=1025.381,-103.616,411.675,166.551,46.198,158.419
C04667=1025.386,-103.367,411.666,166.554,46.195,158.419
C04668=1025.392,-103.117,411.656,166.557,46.192,158.419
C04669=1025.398,-102.867,411.647,166.560,46.190,158.419
C04670=1025.404,-102.618,411.638,166.563,46.187,158.419
C04671=1025.409,-102.368,411.628,166.566,46.184,158.419
C04672=1025.415,-102.118,411.619,166.569,46.181,158.418
C04673=1025.421,-101.868,411.610,166.572,46.178,158.418
C04674=1025.427,-101.618,411.600,166.574,46.175,158.418
C04675=1025.433,-101.333,411.590,166.579,46.172,158.418
C04676=1025.440,-101.046,411.579,166.582,46.169,158.418
C04677=1025.446,-100.761,411.568,166.585,46.166,158.418
C04678=1025.452,-100.475,411.557,166.589,46.163,158.418
C04679=1025.458,-100.225,411.548,166.592,46.160,158.418
C04680=1025.464,-99.975,411.539,166.595,46.157,158.417
C04681=1025.470,-99.725,411.530,166.598,46.154,158.417
C04682=1025.476,-99.476,411.520,166.601,46.151,158.417
C04683=1025.482,-99.226,411.510,166.604,46.148,158.417
C04684=1025.488,-98.976,411.500,166.607,46.146,158.417
C04685=1025.493,-98.727,411.491,166.610,46.143,158.417
C04686=1025.499,-98.477,411.482,166.612,46.140,158.416
C04687=1025.505,-98.226,411.473,166.616,46.137,158.416
C04688=1025.511,-97.977,411.463,166.619,46.134,158.416
C04689=1025.516,-97.727,411.453,166.621,46.131,158.416
C04690=1025.522,-97.477,411.444,166.625,46.129,158.416
C04691=1025.528,-97.227,411.434,166.628,46.126,158.416
C04692=1025.533,-96.978,411.424,166.630,46.123,158.416
C04693=1025.540,-96.728,411.415,166.634,46.121,158.416
C04694=1025.545,-96.478,411.405,166.636,46.118,158.415
C04695=1025.551,-96.229,411.395,166.640,46.115,158.415
C04696=1025.556,-95.979,411.385,166.643,46.113,158.415
C04697=1025.562,-95.729,411.376,166.646,46.110,158.415
C04698=1025.568,-95.479,411.366,166.649,46.107,158.415
C04699=1025.573,-95.230,411.356,166.651,46.105,158.415
C04700=1025.579,-94.980,411.346,166.655,46.102,158.415
C04701=1025.585,-94.730,411.337,166.658,46.099,158.415
C04702=1025.590,-94.480,411.326,166.661,46.097,158.414
C04703=1025.596,-94.231,411.317,166.664,46.094,158.414
C04704=1025.602,-93.981,411.306,166.666,46.091,158.414
C04705=1025.608,-93.732,411.297,166.670,46.089,158.414
C04706=1025.613,-93.482,411.287,166.672,46.086,158.414
C04707=1025.619,-93.232,411.277,166.675,46.083,158.414
C04708=1025.624,-92.982,411.267,166.679,46.081,158.414
C04709=1025.630,-92.733,411.258,166.681,46.078,158.414
C04710=1025.636,-92.483,411.248,166.685,46.075,158.413
C04711=1025.642,-92.233,411.238,166.687,46.073,158.413
C04712=1025.648,-91.983,411.228,166.690,46.070,158.413
C04713=1025.654,-91.733,411.218,166.694,46.067,158.413
C04714=1025.659,-91.484,411.208,166.696,46.065,158.413
C04715=1025.665,-91.234,411.198,166.700,46.062,158.413
C04716=1025.671,-90.984,411.189,166.702,46.059,158.413
C04717=1025.677,-90.735,411.178,166.705,46.057,158.413
C04718=1025.683,-90.485,411.168,166.709,46.054,158.412
C04719=1025.688,-90.235,411.158,166.711,46.051,158.412
C04720=1025.694,-89.985,411.148,166.714,46.048,158.412
C04721=1025.699,-89.736,411.139,166.717,46.046,158.412
C04722=1025.706,-89.487,411.128,166.720,46.043,158.412
C04723=1025.711,-89.236,411.118,166.724,46.040,158.412
C04724=1025.717,-88.987,411.109,166.726,46.038,158.412
C04725=1025.723,-88.737,411.098,166.729,46.035,158.411
C04726=1025.729,-88.487,411.088,166.732,46.032,158.411
C04727=1025.735,-88.237,411.078,166.735,46.030,158.411
C04728=1025.741,-87.987,411.068,166.739,46.027,158.411
C04729=1025.747,-87.738,411.058,166.741,46.024,158.411
C04730=1025.753,-87.488,411.048,166.744,46.021,158.411
C04731=1025.758,-87.238,411.038,166.747,46.019,158.411
C04732=1025.764,-86.989,411.027,166.750,46.016,158.411
C04733=1025.770,-86.740,411.018,166.753,46.013,158.410
C04734=1025.775,-86.489,411.008,166.756,46.011,158.410
C04735=1025.781,-86.240,410.997,166.759,46.008,158.410
C04736=1025.787,-85.990,410.987,166.762,46.005,158.410
C04737=1025.793,-85.740,410.978,166.765,46.002,158.410
C04738=1025.799,-85.491,410.967,166.769,46.000,158.410
C04739=1025.806,-85.206,410.955,166.772,45.997,158.410
C04740=1025.812,-84.923,410.944,166.775,45.993,158.409
C04741=1025.819,-84.639,410.933,166.778,45.990,158.409
C04742=1025.826,-84.355,410.920,166.782,45.987,158.409
C04743=1025.832,-84.105,410.911,166.784,45.984,158.409
C04744=1025.838,-83.855,410.900,166.787,45.982,158.409
C04745=1025.844,-83.606,410.890,166.791,45.979,158.409
C04746=1025.850,-83.356,410.880,166.793,45.976,158.408
C04747=1025.856,-83.106,410.869,166.797,45.974,158.408
C04748=1025.862,-82.856,410.860,166.800,45.971,158.408
C04749=1025.867,-82.607,410.849,166.802,45.968,158.408
C04750=1025.874,-82.357,410.839,166.806,45.965,158.408
C04751=1025.879,-82.108,410.828,166.808,45.963,158.408
C04752=1025.886,-81.858,410.819,166.811,45.960,158.408
C04753=1025.891,-81.608,410.808,166.815,45.957,158.408
C04754=1025.897,-81.359,410.798,166.817,45.954,158.407
C04755=1025.903,-81.109,410.787,166.821,45.952,158.407
C04756=1025.909,-80.859,410.778,166.823,45.949,158.407
C04757=1025.915,-80.610,410.767,166.826,45.946,158.407
C04758=1025.921,-80.359,410.756,166.830,45.943,158.407
C04759=1025.928,-80.110,410.746,166.832,45.941,158.407
C04760=1025.933,-79.860,410.736,166.835,45.938,158.407
C04761=1025.939,-79.610,410.725,166.838,45.935,158.406
C04762=1025.945,-79.361,410.714,166.841,45.933,158.406
C04763=1025.951,-79.111,410.705,166.844,45.930,158.406
C04764=1025.956,-78.861,410.694,166.847,45.928,158.406
C04765=1025.962,-78.612,410.683,166.849,45.925,158.406
C04766=1025.968,-78.362,410.673,166.853,45.922,158.406
C04767=1025.974,-78.112,410.661,166.855,45.920,158.406
C04768=1025.980,-77.862,410.651,166.859,45.917,158.405
C04769=1025.986,-77.613,410.640,166.861,45.915,158.405
C04770=1025.992,-77.363,410.630,166.865,45.912,158.405
C04771=1025.997,-77.113,410.619,166.868,45.909,158.405
C04772=1026.003,-76.864,410.608,166.870,45.907,158.405
C04773=1026.009,-76.614,410.598,166.874,45.904,158.405
C04774=1026.016,-76.364,410.588,166.876,45.902,158.405
C04775=1026.021,-76.114,410.577,166.880,45.899,158.405
C04776=1026.027,-75.865,410.566,166.882,45.896,158.404
C04777=1026.033,-75.615,410.555,166.886,45.894,158.404
C04778=1026.038,-75.365,410.545,166.888,45.891,158.404
C04779=1026.045,-75.115,410.534,166.891,45.889,158.404
C04780=1026.051,-74.866,410.523,166.894,45.886,158.404
C04781=1026.057,-74.616,410.512,166.897,45.883,158.404
C04782=1026.063,-74.367,410.502,166.900,45.881,158.404
C04783=1026.068,-74.117,410.491,166.903,45.878,158.404
C04784=1026.074,-73.867,410.480,166.905,45.876,158.403
C04785=1026.080,-73.617,410.469,166.909,45.873,158.403
C04786=1026.086,-73.368,410.458,166.911,45.871,158.403
C04787=1026.092,-73.118,410.447,166.915,45.869,158.403
C04788=1026.097,-72.868,410.436,166.917,45.866,158.403
C04789=1026.103,-72.618,410.425,166.921,45.864,158.403
C04790=1026.109,-72.369,410.414,166.923,45.861,158.403
C04791=1026.114,-72.119,410.403,166.926,45.859,158.403
C04792=1026.120,-71.870,410.392,166.929,45.856,158.403
C04793=1026.126,-71.620,410.381,166.932,45.854,158.402
C04794=1026.132,-71.370,410.370,166.935,45.852,158.402
C04795=1026.138,-71.121,410.359,166.937,45.849,158.402
C04796=1026.143,-70.871,410.348,166.941,45.847,158.402
C04797=1026.149,-70.621,410.336,166.943,45.844,158.402
C04798=1026.155,-70.371,410.326,166.947,45.842,158.402
C04799=1026.161,-70.122,410.314,166.949,45.839,158.402
C04800=1026.167,-69.873,410.303,166.953,45.837,158.402
C04801=1026.173,-69.623,410.292,166.955,45.834,158.402
C04802=1026.179,-69.373,410.281,166.958,45.832,158.401
C04803=1026.185,-69.091,410.268,166.961,45.829,158.401
C04804=1026.192,-68.809,410.256,166.965,45.827,158.401
C04805=1026.198,-68.528,410.243,166.968,45.824,158.401
C04806=1026.205,-68.246,410.231,166.971,45.821,158.401
C04807=1026.211,-67.996,410.219,166.975,45.818,158.401
C04808=1026.217,-67.746,410.208,166.977,45.816,158.401
C04809=1026.222,-67.497,410.197,166.980,45.814,158.401
C04810=1026.229,-67.247,410.186,166.983,45.811,158.400
C04811=1026.235,-66.998,410.174,166.985,45.809,158.400
C04812=1026.240,-66.748,410.164,166.989,45.806,158.400
C04813=1026.246,-66.498,410.152,166.991,45.804,158.400
C04814=1026.252,-66.248,410.141,166.995,45.801,158.400
C04815=1026.258,-65.999,410.130,166.997,45.799,158.400
C04816=1026.264,-65.749,410.118,167.001,45.796,158.400
C04817=1026.270,-65.500,410.107,167.003,45.793,158.400
C04818=1026.276,-65.250,410.096,167.005,45.791,158.399
C04819=1026.282,-65.000,410.085,167.009,45.788,158.399
C04820=1026.287,-64.750,410.074,167.011,45.786,158.399
C04821=1026.294,-64.501,410.062,167.015,45.783,158.399
C04822=1026.299,-64.251,410.051,167.017,45.781,158.399
C04823=1026.306,-64.001,410.039,167.021,45.778,158.399
C04824=1026.311,-63.752,410.029,167.023,45.776,158.399
C04825=1026.318,-63.503,410.017,167.027,45.773,158.399
C04826=1026.323,-63.252,410.005,167.029,45.771,158.398
C04827=1026.329,-63.003,409.994,167.033,45.768,158.398
C04828=1026.336,-62.753,409.982,167.035,45.766,158.398
C04829=1026.341,-62.504,409.971,167.037,45.764,158.398
C04830=1026.348,-62.254,409.960,167.041,45.761,158.398
C04831=1026.354,-62.005,409.949,167.043,45.759,158.398
C04832=1026.359,-61.754,409.937,167.047,45.756,158.398
C04833=1026.365,-61.505,409.926,167.049,45.754,158.398
C04834=1026.371,-61.256,409.914,167.053,45.751,158.398
C04835=1026.377,-61.006,409.903,167.055,45.749,158.397
C04836=1026.383,-60.756,409.892,167.058,45.746,158.397
C04837=1026.389,-60.506,409.880,167.061,45.744,158.397
C04838=1026.395,-60.257,409.869,167.064,45.741,158.397
C04839=1026.401,-60.007,409.857,167.067,45.739,158.397
C04840=1026.407,-59.758,409.846,167.070,45.736,158.397
C04841=1026.413,-59.507,409.835,167.073,45.734,158.397
C04842=1026.419,-59.258,409.823,167.075,45.731,158.396
C04843=1026.425,-59.008,409.811,167.078,45.728,158.396
C04844=1026.432,-58.759,409.799,167.081,45.726,158.396
C04845=1026.438,-58.509,409.788,167.084,45.723,158.396
C04846=1026.444,-58.259,409.776,167.087,45.721,158.396
C04847=1026.449,-58.010,409.765,167.090,45.718,158.396
C04848=1026.455,-57.759,409.754,167.093,45.716,158.396
C04849=1026.462,-57.511,409.742,167.096,45.713,158.396
C04850=1026.468,-57.260,409.731,167.099,45.711,158.395
C04851=1026.474,-57.012,409.719,167.102,45.708,158.395
C04852=1026.480,-56.761,409.707,167.104,45.705,158.395
C04853=1026.486,-56.511,409.696,167.107,45.703,158.395
C04854=1026.492,-56.262,409.685,167.110,45.700,158.395
C04855=1026.499,-56.012,409.673,167.113,45.698,158.395
C04856=1026.505,-55.764,409.661,167.116,45.695,158.395
C04857=1026.510,-55.513,409.649,167.119,45.693,158.394
C04858=1026.517,-55.263,409.637,167.122,45.690,158.394
C04859=1026.523,-55.014,409.626,167.124,45.687,158.394
C04860=1026.529,-54.764,409.614,167.128,45.685,158.394
C04861=1026.535,-54.514,409.603,167.130,45.682,158.394
C04862=1026.541,-54.265,409.591,167.133,45.680,158.394
C04863=1026.547,-54.015,409.580,167.136,45.677,158.394
C04864=1026.554,-53.765,409.568,167.139,45.675,158.393
C04865=1026.560,-53.516,409.556,167.142,45.672,158.393
C04866=1026.566,-53.266,409.544,167.144,45.670,158.393
C04867=1026.572,-52.986,409.531,167.147,45.667,158.393
C04868=1026.580,-52.705,409.519,167.151,45.664,158.393
C04869=1026.587,-52.425,409.505,167.154,45.661,158.393
C04870=1026.593,-52.144,409.492,167.158,45.658,158.393
C04871=1026.600,-51.895,409.480,167.160,45.656,158.392
C04872=1026.606,-51.645,409.468,167.163,45.653,158.392
C04873=1026.613,-51.395,409.457,167.166,45.651,158.392
C04874=1026.618,-51.146,409.445,167.169,45.648,158.392
C04875=1026.625,-50.896,409.433,167.172,45.646,158.392
C04876=1026.631,-50.647,409.421,167.175,45.643,158.392
C04877=1026.636,-50.397,409.409,167.178,45.641,158.392
C04878=1026.642,-50.147,409.397,167.180,45.638,158.391
C04879=1026.649,-49.897,409.385,167.184,45.636,158.391
C04880=1026.655,-49.647,409.372,167.186,45.634,158.391
C04881=1026.661,-49.399,409.361,167.188,45.631,158.391
C04882=1026.666,-49.148,409.349,167.192,45.629,158.391
C04883=1026.672,-48.898,409.336,167.195,45.627,158.391
C04884=1026.678,-48.649,409.325,167.197,45.624,158.391
C04885=1026.684,-48.399,409.312,167.200,45.622,158.391
C04886=1026.690,-48.149,409.300,167.203,45.620,158.391
C04887=1026.697,-47.900,409.288,167.205,45.617,158.390
C04888=1026.702,-47.651,409.275,167.209,45.615,158.390
C04889=1026.709,-47.401,409.264,167.211,45.612,158.390
C04890=1026.715,-47.151,409.251,167.214,45.610,158.390
C04891=1026.720,-46.902,409.239,167.217,45.608,158.390
C04892=1026.727,-46.653,409.227,167.220,45.605,158.390
C04893=1026.732,-46.403,409.214,167.222,45.603,158.390
C04894=1026.738,-46.153,409.202,167.226,45.600,158.389
C04895=1026.745,-45.903,409.190,167.228,45.598,158.389
C04896=1026.750,-45.654,409.178,167.231,45.596,158.389
C04897=1026.757,-45.404,409.166,167.234,45.593,158.389
C04898=1026.763,-45.154,409.154,167.237,45.591,158.389
C04899=1026.768,-44.904,409.141,167.239,45.589,158.389
C04900=1026.775,-44.656,409.129,167.242,45.586,158.389
C04901=1026.781,-44.406,409.116,167.245,45.584,158.389
C04902=1026.787,-44.156,409.104,167.247,45.581,158.388
C04903=1026.793,-43.906,409.092,167.251,45.579,158.388
C04904=1026.799,-43.657,409.079,167.253,45.576,158.388
C04905=1026.805,-43.407,409.067,167.257,45.574,158.388
C04906=1026.811,-43.158,409.055,167.259,45.572,158.388
C04907=1026.817,-42.908,409.043,167.262,45.569,158.388
C04908=1026.823,-42.658,409.030,167.265,45.567,158.388
C04909=1026.830,-42.408,409.018,167.268,45.564,158.388
C04910=1026.836,-42.159,409.005,167.270,45.562,158.387
C04911=1026.842,-41.909,408.994,167.274,45.559,158.387
C04912=1026.848,-41.659,408.981,167.276,45.557,158.387
C04913=1026.853,-41.410,408.969,167.279,45.555,158.387
C04914=1026.860,-41.161,408.956,167.282,45.552,158.387
C04915=1026.866,-40.911,408.944,167.285,45.550,158.387
C04916=1026.872,-40.661,408.931,167.287,45.547,158.387
C04917=1026.879,-40.412,408.919,167.290,45.545,158.387
C04918=1026.885,-40.162,408.907,167.293,45.542,158.386
C04919=1026.891,-39.912,408.894,167.295,45.540,158.386
C04920=1026.897,-39.662,408.882,167.299,45.538,158.386
C04921=1026.903,-39.413,408.869,167.301,45.535,158.386
C04922=1026.909,-39.163,408.856,167.303,45.533,158.386
C04923=1026.915,-38.914,408.844,167.307,45.531,158.386
C04924=1026.921,-38.664,408.832,167.310,45.528,158.386
C04925=1026.928,-38.415,408.819,167.312,45.526,158.386
C04926=1026.933,-38.165,408.806,167.315,45.524,158.385
C04927=1026.939,-37.915,408.794,167.318,45.521,158.385
C04928=1026.945,-37.666,408.781,167.321,45.519,158.385
C04929=1026.951,-37.416,408.768,167.323,45.517,158.385
C04930=1026.957,-37.166,408.755,167.327,45.514,158.385
C04931=1026.964,-36.886,408.740,167.329,45.512,158.385
C04932=1026.971,-36.606,408.727,167.332,45.510,158.385
C04933=1026.978,-36.326,408.712,167.336,45.507,158.384
C04934=1026.984,-36.045,408.698,167.338,45.505,158.384
C04935=1026.991,-35.796,408.685,167.342,45.502,158.384
C04936=1026.997,-35.546,408.672,167.344,45.500,158.384
C04937=1027.003,-35.297,408.661,167.347,45.498,158.384
C04938=1027.009,-35.048,408.647,167.349,45.495,158.384
C04939=1027.015,-34.798,408.635,167.353,45.493,158.384
C04940=1027.021,-34.549,408.621,167.355,45.491,158.384
C04941=1027.027,-34.299,408.609,167.358,45.488,158.383
C04942=1027.033,-34.050,408.596,167.360,45.486,158.383
C04943=1027.039,-33.800,408.583,167.364,45.484,158.383
C04944=1027.045,-33.550,408.571,167.366,45.481,158.383
C04945=1027.051,-33.301,408.557,167.369,45.479,158.383
C04946=1027.057,-33.051,408.545,167.371,45.477,158.383
C04947=1027.064,-32.801,408.531,167.374,45.474,158.383
C04948=1027.070,-32.551,408.518,167.377,45.472,158.383
C04949=1027.076,-32.302,408.505,167.379,45.469,158.382
C04950=1027.082,-32.052,408.493,167.383,45.467,158.382
C04951=1027.088,-31.803,408.479,167.386,45.465,158.382
C04952=1027.094,-31.553,408.467,167.388,45.462,158.382
C04953=1027.100,-31.304,408.454,167.390,45.460,158.382
C04954=1027.107,-31.054,408.442,167.394,45.458,158.382
C04955=1027.113,-30.805,408.428,167.396,45.455,158.382
C04956=1027.119,-30.555,408.416,167.399,45.453,158.382
C04957=1027.125,-30.306,408.403,167.401,45.450,158.381
C04958=1027.131,-30.056,408.390,167.405,45.448,158.381
C04959=1027.137,-29.806,408.377,167.407,45.446,158.381
C04960=1027.144,-29.557,408.363,167.410,45.444,158.381
C04961=1027.149,-29.307,408.351,167.413,45.441,158.381
C04962=1027.156,-29.057,408.337,167.416,45.439,158.381
C04963=1027.162,-28.807,408.325,167.418,45.437,158.381
C04964=1027.168,-28.558,408.311,167.421,45.435,158.380
C04965=1027.175,-28.309,408.298,167.424,45.432,158.380
C04966=1027.180,-28.059,408.286,167.427,45.430,158.380
C04967=1027.187,-27.810,408.272,167.429,45.427,158.380
C04968=1027.193,-27.560,408.260,167.431,45.425,158.380
C04969=1027.199,-27.311,408.247,167.435,45.423,158.380
C04970=1027.206,-27.061,408.233,167.437,45.420,158.380
C04971=1027.212,-26.811,408.220,167.440,45.418,158.379
C04972=1027.217,-26.561,408.206,167.442,45.416,158.379
C04973=1027.223,-26.312,408.193,167.445,45.414,158.379
C04974=1027.229,-26.063,408.180,167.448,45.411,158.379
C04975=1027.236,-25.813,408.167,167.451,45.409,158.379
C04976=1027.241,-25.563,408.153,167.453,45.407,158.379
C04977=1027.248,-25.313,408.140,167.456,45.405,158.379
C04978=1027.254,-25.064,408.127,167.458,45.402,158.379
C04979=1027.260,-24.815,408.113,167.462,45.400,158.379
C04980=1027.266,-24.566,408.100,167.465,45.398,158.378
C04981=1027.271,-24.315,408.087,167.467,45.395,158.378
C04982=1027.278,-24.066,408.074,167.469,45.393,158.378
C04983=1027.284,-23.816,408.060,167.472,45.391,158.378
C04984=1027.291,-23.567,408.047,167.476,45.389,158.378
C04985=1027.296,-23.317,408.033,167.478,45.386,158.378
C04986=1027.302,-23.068,408.020,167.480,45.384,158.378
C04987=1027.308,-22.818,408.007,167.483,45.382,158.378
C04988=1027.315,-22.568,407.993,167.485,45.379,158.377
C04989=1027.321,-22.319,407.980,167.489,45.377,158.377
C04990=1027.327,-22.069,407.966,167.491,45.375,158.377
C04991=1027.333,-21.820,407.953,167.494,45.373,158.377
C04992=1027.339,-21.571,407.940,167.496,45.371,158.377
C04993=1027.345,-21.320,407.926,167.499,45.369,158.377
C04994=1027.352,-21.071,407.912,167.503,45.366,158.377
C04995=1027.359,-20.790,407.898,167.505,45.364,158.376
C04996=1027.365,-20.509,407.882,167.508,45.361,158.376
C04997=1027.372,-20.228,407.867,167.511,45.359,158.376
C04998=1027.379,-19.947,407.852,167.514,45.356,158.376
C04999=1027.385,-19.697,407.838,167.517,45.354,158.376
C05000=1027.391,-19.448,407.825,167.519,45.351,158.376
C05001=1027.397,-19.199,407.812,167.523,45.349,158.376
C05002=1027.404,-18.949,407.798,167.525,45.347,158.375
C05003=1027.410,-18.699,407.784,167.527,45.344,158.375
C05004=1027.416,-18.450,407.771,167.530,45.342,158.375
C05005=1027.423,-18.200,407.757,167.533,45.340,158.375
C05006=1027.429,-17.951,407.744,167.536,45.337,158.375
C05007=1027.434,-17.701,407.730,167.538,45.335,158.375
C05008=1027.441,-17.451,407.717,167.541,45.333,158.375
C05009=1027.447,-17.202,407.703,167.543,45.330,158.374
C05010=1027.453,-16.952,407.690,167.546,45.328,158.374
C05011=1027.460,-16.702,407.676,167.549,45.326,158.374
C05012=1027.466,-16.453,407.663,167.552,45.323,158.374
C05013=1027.472,-16.204,407.649,167.554,45.321,158.374
C05014=1027.479,-15.954,407.634,167.557,45.319,158.374
C05015=1027.485,-15.705,407.621,167.559,45.317,158.374
C05016=1027.491,-15.456,407.608,167.562,45.315,158.373
C05017=1027.497,-15.205,407.594,167.565,45.313,158.373
C05018=1027.503,-14.956,407.580,167.568,45.310,158.373
C05019=1027.509,-14.707,407.567,167.570,45.308,158.373
C05020=1027.515,-14.456,407.552,167.573,45.306,158.373
C05021=1027.521,-14.208,407.538,167.575,45.304,158.373
C05022=1027.527,-13.958,407.524,167.578,45.301,158.373
C05023=1027.534,-13.708,407.511,167.580,45.299,158.373
C05024=1027.539,-13.459,407.497,167.584,45.297,158.373
C05025=1027.546,-13.210,407.483,167.586,45.295,158.372
C05026=1027.552,-12.960,407.469,167.589,45.293,158.372
C05027=1027.558,-12.710,407.455,167.591,45.290,158.372
C05028=1027.564,-12.460,407.441,167.594,45.288,158.372
C05029=1027.571,-12.211,407.427,167.596,45.286,158.372
C05030=1027.576,-11.962,407.413,167.599,45.284,158.372
C05031=1027.583,-11.712,407.400,167.601,45.281,158.371
C05032=1027.588,-11.462,407.386,167.605,45.279,158.371
C05033=1027.595,-11.213,407.371,167.608,45.277,158.371
C05034=1027.601,-10.963,407.358,167.610,45.275,158.371
C05035=1027.606,-10.714,407.344,167.612,45.272,158.371
C05036=1027.613,-10.464,407.329,167.615,45.270,158.371
C05037=1027.619,-10.215,407.316,167.618,45.268,158.371
C05038=1027.626,-9.965,407.302,167.620,45.266,158.371
C05039=1027.632,-9.716,407.287,167.622,45.264,158.370
C05040=1027.638,-9.466,407.274,167.626,45.262,158.370
C05041=1027.644,-9.216,407.260,167.629,45.260,158.370
C05042=1027.650,-8.968,407.246,167.631,45.257,158.370
C05043=1027.656,-8.718,407.232,167.633,45.255,158.370
C05044=1027.662,-8.468,407.218,167.636,45.253,158.370
C05045=1027.669,-8.219,407.203,167.638,45.250,158.370
C05046=1027.675,-7.969,407.190,167.641,45.248,158.370
C05047=1027.682,-7.720,407.175,167.643,45.246,158.369
C05048=1027.687,-7.470,407.161,167.647,45.243,158.369
C05049=1027.694,-7.220,407.148,167.649,45.241,158.369
C05050=1027.700,-6.971,407.133,167.652,45.239,158.369
C05051=1027.706,-6.721,407.119,167.654,45.237,158.369
C05052=1027.712,-6.472,407.105,167.657,45.235,158.369
C05053=1027.718,-6.222,407.091,167.659,45.233,158.369
C05054=1027.725,-5.973,407.077,167.662,45.230,158.368
C05055=1027.731,-5.723,407.062,167.664,45.228,158.368
C05056=1027.737,-5.474,407.049,167.668,45.226,158.368
C05057=1027.744,-5.224,407.034,167.670,45.223,158.368
C05058=1027.749,-4.975,407.020,167.673,45.221,158.368
C05059=1027.757,-4.692,407.004,167.675,45.218,158.368
C05060=1027.764,-4.409,406.988,167.679,45.216,158.368
C05061=1027.771,-4.127,406.973,167.681,45.213,158.367
C05062=1027.778,-3.845,406.956,167.684,45.210,158.367
C05063=1027.784,-3.595,406.941,167.687,45.208,158.367
C05064=1027.790,-3.345,406.927,167.689,45.206,158.367
C05065=1027.796,-3.096,406.912,167.692,45.204,158.367
C05066=1027.803,-2.846,406.898,167.695,45.202,158.367
C05067=1027.808,-2.597,406.884,167.697,45.200,158.367
C05068=1027.815,-2.347,406.869,167.700,45.198,158.366
C05069=1027.820,-2.098,406.855,167.702,45.196,158.366
C05070=1027.827,-1.848,406.840,167.705,45.194,158.366
C05071=1027.833,-1.599,406.826,167.707,45.192,158.366
C05072=1027.839,-1.349,406.811,167.710,45.190,158.366
C05073=1027.844,-1.100,406.797,167.712,45.188,158.366
C05074=1027.851,-0.850,406.782,167.715,45.186,158.366
C05075=1027.857,-0.601,406.767,167.717,45.183,158.365
C05076=1027.863,-0.351,406.753,167.721,45.181,158.365
C05077=1027.869,-0.101,406.738,167.723,45.179,158.365
C05078=1027.876,0.147,406.724,167.726,45.177,158.365
C05079=1027.882,0.397,406.709,167.729,45.175,158.365
C05080=1027.887,0.647,406.695,167.731,45.173,158.365
C05081=1027.894,0.896,406.680,167.733,45.170,158.365
C05082=1027.900,1.146,406.665,167.736,45.168,158.365
C05083=1027.906,1.395,406.651,167.739,45.166,158.364
C05084=1027.912,1.645,406.637,167.741,45.164,158.364
C05085=1027.918,1.894,406.622,167.744,45.162,158.364
C05086=1027.924,2.144,406.607,167.746,45.160,158.364
C05087=1027.931,2.393,406.592,167.749,45.158,158.364
C05088=1027.936,2.642,406.577,167.751,45.156,158.364
C05089=1027.942,2.893,406.563,167.754,45.154,158.364
C05090=1027.949,3.142,406.548,167.756,45.151,158.363
C05091=1027.955,3.391,406.534,167.759,45.149,158.363
C05092=1027.961,3.641,406.519,167.761,45.147,158.363
C05093=1027.967,3.891,406.504,167.764,45.145,158.363
C05094=1027.973,4.140,406.489,167.766,45.143,158.363
C05095=1027.980,4.389,406.475,167.769,45.140,158.363
C05096=1027.986,4.639,406.461,167.771,45.138,158.363
C05097=1027.992,4.888,406.446,167.774,45.136,158.363
C05098=1027.998,5.138,406.431,167.776,45.134,158.362
C05099=1028.005,5.387,406.416,167.779,45.132,158.362
C05100=1028.011,5.636,406.402,167.781,45.130,158.362
C05101=1028.017,5.886,406.387,167.785,45.127,158.362
C05102=1028.023,6.136,406.372,167.787,45.125,158.362
C05103=1028.029,6.385,406.357,167.790,45.123,158.362
C05104=1028.036,6.634,406.342,167.792,45.121,158.362
C05105=1028.042,6.884,406.327,167.795,45.119,158.361
C05106=1028.048,7.134,406.312,167.797,45.116,158.361
C05107=1028.054,7.383,406.298,167.800,45.114,158.361
C05108=1028.060,7.633,406.283,167.802,45.112,158.361
C05109=1028.067,7.883,406.269,167.805,45.110,158.361
C05110=1028.072,8.131,406.254,167.807,45.107,158.361
C05111=1028.079,8.381,406.239,167.810,45.105,158.361
C05112=1028.085,8.631,406.224,167.812,45.103,158.360
C05113=1028.092,8.880,406.209,167.815,45.101,158.360
C05114=1028.098,9.130,406.194,167.817,45.099,158.360
C05115=1028.104,9.379,406.180,167.820,45.097,158.360
C05116=1028.110,9.629,406.165,167.822,45.094,158.360
C05117=1028.116,9.878,406.150,167.825,45.092,158.360
C05118=1028.123,10.128,406.135,167.827,45.090,158.359
C05119=1028.129,10.377,406.120,167.830,45.087,158.359
C05120=1028.135,10.626,406.105,167.832,45.085,158.359
C05121=1028.142,10.876,406.090,167.835,45.083,158.359
C05122=1028.148,11.125,406.075,167.837,45.081,158.359
C05123=1028.155,11.410,406.059,167.841,45.079,158.359
C05124=1028.162,11.695,406.041,167.843,45.076,158.358
C05125=1028.170,11.979,406.025,167.846,45.073,158.358
C05126=1028.177,12.263,406.007,167.849,45.071,158.358
C05127=1028.183,12.513,405.992,167.851,45.068,158.358
C05128=1028.190,12.763,405.977,167.854,45.066,158.358
C05129=1028.196,13.012,405.962,167.857,45.064,158.358
C05130=1028.202,13.261,405.947,167.860,45.061,158.357
C05131=1028.209,13.510,405.932,167.862,45.060,158.357
C05132=1028.215,13.760,405.917,167.865,45.058,158.357
C05133=1028.221,14.010,405.902,167.867,45.055,158.357
C05134=1028.227,14.260,405.887,167.870,45.053,158.357
C05135=1028.233,14.509,405.872,167.872,45.051,158.357
C05136=1028.239,14.758,405.857,167.875,45.049,158.357
C05137=1028.246,15.007,405.842,167.877,45.047,158.357
C05138=1028.252,15.257,405.826,167.880,45.044,158.356
C05139=1028.258,15.507,405.811,167.882,45.042,158.356
C05140=1028.265,15.756,405.795,167.885,45.040,158.356
C05141=1028.270,16.006,405.780,167.888,45.038,158.356
C05142=1028.277,16.256,405.765,167.890,45.036,158.356
C05143=1028.283,16.504,405.750,167.891,45.034,158.355
C05144=1028.289,16.754,405.735,167.894,45.032,158.355
C05145=1028.295,17.004,405.719,167.897,45.030,158.355
C05146=1028.301,17.253,405.704,167.899,45.028,158.355
C05147=1028.308,17.502,405.689,167.901,45.025,158.355
C05148=1028.314,17.752,405.674,167.904,45.023,158.355
C05149=1028.320,18.001,405.657,167.907,45.021,158.355
C05150=1028.327,18.251,405.642,167.909,45.019,158.354
C05151=1028.332,18.500,405.628,167.911,45.017,158.354
C05152=1028.339,18.749,405.612,167.914,45.015,158.354
C05153=1028.345,18.999,405.597,167.917,45.013,158.354
C05154=1028.351,19.248,405.582,167.919,45.010,158.354
C05155=1028.358,19.498,405.566,167.922,45.008,158.354
C05156=1028.363,19.747,405.550,167.924,45.006,158.354
C05157=1028.370,19.997,405.535,167.927,45.004,158.353
C05158=1028.376,20.246,405.520,167.929,45.002,158.353
C05159=1028.382,20.496,405.504,167.932,44.999,158.353
C05160=1028.389,20.745,405.489,167.934,44.997,158.353
C05161=1028.394,20.995,405.473,167.937,44.995,158.353
C05162=1028.401,21.244,405.457,167.939,44.993,158.353
C05163=1028.407,21.494,405.442,167.942,44.991,158.353
C05164=1028.413,21.742,405.427,167.944,44.989,158.352
C05165=1028.419,21.992,405.412,167.947,44.987,158.352
C05166=1028.425,22.242,405.395,167.949,44.985,158.352
C05167=1028.432,22.491,405.380,167.952,44.983,158.352
C05168=1028.438,22.741,405.364,167.954,44.980,158.352
C05169=1028.444,22.990,405.349,167.957,44.978,158.352
C05170=1028.450,23.240,405.333,167.959,44.976,158.352
C05171=1028.456,23.489,405.318,167.962,44.974,158.351
C05172=1028.463,23.738,405.302,167.964,44.972,158.351
C05173=1028.469,23.988,405.286,167.967,44.970,158.351
C05174=1028.475,24.237,405.271,167.969,44.968,158.351
C05175=1028.481,24.487,405.255,167.972,44.966,158.351
C05176=1028.488,24.736,405.240,167.973,44.963,158.351
C05177=1028.494,24.986,405.224,167.976,44.961,158.350
C05178=1028.500,25.235,405.209,167.978,44.959,158.350
C05179=1028.507,25.484,405.193,167.981,44.957,158.350
C05180=1028.513,25.734,405.177,167.983,44.955,158.350
C05181=1028.519,25.983,405.162,167.986,44.953,158.350
C05182=1028.525,26.233,405.146,167.988,44.951,158.350
C05183=1028.531,26.482,405.131,167.991,44.949,158.350
C05184=1028.537,26.732,405.114,167.993,44.946,158.349
C05185=1028.544,26.981,405.099,167.996,44.944,158.349
C05186=1028.550,27.231,405.083,167.999,44.942,158.349
C05187=1028.558,27.517,405.065,168.001,44.939,158.349
C05188=1028.564,27.802,405.047,168.004,44.937,158.349
C05189=1028.571,28.088,405.029,168.007,44.935,158.349
C05190=1028.579,28.374,405.010,168.010,44.932,158.348
C05191=1028.585,28.624,404.995,168.012,44.930,158.348
C05192=1028.591,28.873,404.979,168.014,44.928,158.348
C05193=1028.597,29.122,404.963,168.017,44.926,158.348
C05194=1028.604,29.371,404.947,168.019,44.924,158.348
C05195=1028.609,29.621,404.931,168.022,44.922,158.348
C05196=1028.615,29.871,404.915,168.025,44.920,158.348
C05197=1028.622,30.120,404.899,168.027,44.917,158.347
C05198=1028.628,30.369,404.883,168.029,44.915,158.347
C05199=1028.634,30.618,404.867,168.032,44.913,158.347
C05200=1028.640,30.868,404.852,168.035,44.911,158.347
C05201=1028.646,31.117,404.836,168.037,44.909,158.347
C05202=1028.652,31.367,404.819,168.040,44.907,158.347
C05203=1028.659,31.616,404.804,168.041,44.905,158.346
C05204=1028.665,31.865,404.788,168.044,44.903,158.346
C05205=1028.671,32.115,404.771,168.046,44.901,158.346
C05206=1028.678,32.364,404.755,168.049,44.898,158.346
C05207=1028.684,32.614,404.740,168.051,44.896,158.346
C05208=1028.690,32.863,404.723,168.054,44.895,158.346
C05209=1028.696,33.113,404.707,168.056,44.893,158.346
C05210=1028.702,33.362,404.692,168.059,44.891,158.345
C05211=1028.708,33.611,404.675,168.061,44.888,158.345
C05212=1028.714,33.861,404.659,168.064,44.886,158.345
C05213=1028.721,34.110,404.643,168.066,44.884,158.345
C05214=1028.727,34.360,404.627,168.069,44.882,158.345
C05215=1028.733,34.609,404.611,168.071,44.879,158.345
C05216=1028.740,34.858,404.595,168.073,44.878,158.344
C05217=1028.746,35.108,404.579,168.075,44.876,158.344
C05218=1028.752,35.357,404.563,168.078,44.874,158.344
C05219=1028.758,35.606,404.547,168.080,44.871,158.344
C05220=1028.765,35.856,404.531,168.083,44.869,158.344
C05221=1028.771,36.106,404.515,168.085,44.867,158.344
C05222=1028.777,36.355,404.498,168.088,44.864,158.343
C05223=1028.783,36.604,404.483,168.090,44.862,158.343
C05224=1028.789,36.853,404.466,168.093,44.860,158.343
C05225=1028.795,37.103,404.450,168.095,44.859,158.343
C05226=1028.802,37.353,404.433,168.098,44.856,158.343
C05227=1028.808,37.582,404.418,168.099,44.854,158.343
C05228=1028.813,37.811,404.404,168.102,44.853,158.343
C05229=1028.819,38.040,404.389,168.105,44.851,158.343
C05230=1028.824,38.271,404.373,168.106,44.849,158.342
C05231=1028.830,38.500,404.358,168.109,44.847,158.342
C05232=1028.836,38.729,404.344,168.111,44.845,158.342
C05233=1028.842,38.958,404.328,168.113,44.843,158.342
C05234=1028.848,39.189,404.314,168.116,44.841,158.342
C05235=1028.854,39.438,404.297,168.118,44.839,158.342
C05236=1028.860,39.687,404.280,168.121,44.837,158.341
C05237=1028.866,39.936,404.264,168.123,44.835,158.341
C05238=1028.872,40.185,404.248,168.126,44.833,158.341
C05239=1028.878,40.435,404.231,168.127,44.831,158.341
C05240=1028.884,40.685,404.215,168.130,44.828,158.341
C05241=1028.890,40.934,404.199,168.132,44.826,158.341
C05242=1028.897,41.183,404.182,168.135,44.825,158.341
C05243=1028.903,41.432,404.165,168.137,44.823,158.340
C05244=1028.909,41.682,404.149,168.140,44.821,158.340
C05245=1028.915,41.932,404.133,168.142,44.818,158.340
C05246=1028.921,42.181,404.116,168.145,44.816,158.340
C05247=1028.927,42.430,404.100,168.147,44.814,158.340
C05248=1028.934,42.680,404.083,168.149,44.812,158.340
C05249=1028.940,42.929,404.067,168.151,44.810,158.339
C05250=1028.946,43.178,404.050,168.154,44.808,158.339
C05251=1028.954,43.504,404.028,168.157,44.805,158.339
C05252=1028.962,43.829,404.006,168.161,44.803,158.339
C05253=1028.970,44.156,403.985,168.163,44.800,158.339
C05254=1028.977,44.481,403.963,168.167,44.798,158.339
C05255=1028.983,44.730,403.947,168.169,44.796,158.339
C05256=1028.990,44.980,403.929,168.172,44.794,158.338
C05257=1028.996,45.229,403.913,168.173,44.791,158.338
C05258=1029.002,45.478,403.896,168.176,44.789,158.338
C05259=1029.007,45.727,403.879,168.178,44.788,158.338
C05260=1029.014,45.977,403.862,168.181,44.786,158.338
C05261=1029.020,46.226,403.845,168.183,44.784,158.338
C05262=1029.026,46.476,403.829,168.186,44.782,158.337
C05263=1029.033,46.725,403.812,168.189,44.780,158.337
C05264=1029.038,46.975,403.795,168.190,44.778,158.337
C05265=1029.044,47.224,403.779,168.193,44.776,158.337
C05266=1029.050,47.473,403.762,168.195,44.774,158.337
C05267=1029.057,47.723,403.745,168.198,44.771,158.337
C05268=1029.063,47.972,403.728,168.200,44.769,158.337
C05269=1029.069,48.221,403.711,168.203,44.767,158.336
C05270=1029.075,48.471,403.694,168.204,44.766,158.336
C05271=1029.081,48.720,403.678,168.207,44.764,158.336
C05272=1029.088,48.969,403.661,168.210,44.762,158.336
C05273=1029.093,49.219,403.644,168.212,44.760,158.336
C05274=1029.100,49.468,403.627,168.214,44.757,158.336
C05275=1029.106,49.717,403.610,168.217,44.755,158.335
C05276=1029.112,49.967,403.593,168.220,44.753,158.335
C05277=1029.118,50.216,403.576,168.221,44.751,158.335
C05278=1029.124,50.465,403.559,168.224,44.750,158.335
C05279=1029.130,50.715,403.543,168.226,44.748,158.335
C05280=1029.137,50.964,403.526,168.229,44.745,158.335
C05281=1029.142,51.213,403.509,168.231,44.743,158.335
C05282=1029.149,51.463,403.491,168.234,44.741,158.334
C05283=1029.155,51.712,403.475,168.236,44.739,158.334
C05284=1029.162,51.962,403.458,168.239,44.737,158.334
C05285=1029.167,52.211,403.441,168.240,44.735,158.334
C05286=1029.173,52.460,403.424,168.243,44.733,158.334
C05287=1029.180,52.710,403.407,168.245,44.731,158.334
C05288=1029.186,52.959,403.390,168.248,44.729,158.334
C05289=1029.191,53.208,403.373,168.251,44.727,158.333
C05290=1029.198,53.458,403.356,168.253,44.725,158.333
C05291=1029.204,53.707,403.339,168.255,44.722,158.333
C05292=1029.211,53.957,403.323,168.257,44.720,158.333
C05293=1029.216,54.206,403.305,168.260,44.719,158.333
C05294=1029.223,54.455,403.288,168.262,44.717,158.333
C05295=1029.229,54.704,403.271,168.265,44.714,158.332
C05296=1029.235,54.953,403.254,168.267,44.712,158.332
C05297=1029.241,55.203,403.237,168.270,44.710,158.332
C05298=1029.247,55.452,403.220,168.272,44.708,158.332
C05299=1029.254,55.702,403.203,168.275,44.706,158.332
C05300=1029.261,55.950,403.186,168.276,44.704,158.331
C05301=1029.266,56.201,403.169,168.279,44.702,158.331
C05302=1029.273,56.449,403.152,168.281,44.700,158.331
C05303=1029.279,56.699,403.134,168.284,44.698,158.331
C05304=1029.285,56.948,403.118,168.286,44.695,158.331
C05305=1029.292,57.198,403.100,168.289,44.693,158.331
C05306=1029.298,57.447,403.083,168.291,44.691,158.331
C05307=1029.304,57.697,403.067,168.294,44.689,158.330
C05308=1029.311,57.946,403.050,168.296,44.687,158.330
C05309=1029.317,58.195,403.032,168.298,44.685,158.330
C05310=1029.323,58.444,403.015,168.300,44.683,158.330
C05311=1029.330,58.694,402.998,168.303,44.680,158.330
C05312=1029.335,58.943,402.981,168.305,44.678,158.329
C05313=1029.342,59.193,402.963,168.308,44.676,158.329
C05314=1029.348,59.441,402.946,168.311,44.675,158.329
C05315=1029.355,59.727,402.926,168.313,44.672,158.329
C05316=1029.363,60.013,402.907,168.316,44.669,158.329
C05317=1029.369,60.298,402.887,168.319,44.667,158.329
C05318=1029.377,60.584,402.868,168.321,44.664,158.328
C05319=1029.384,60.833,402.851,168.324,44.663,158.328
C05320=1029.389,61.082,402.833,168.326,44.660,158.328
C05321=1029.396,61.332,402.816,168.329,44.658,158.328
C05322=1029.402,61.581,402.800,168.331,44.656,158.328
C05323=1029.409,61.830,402.782,168.334,44.653,158.327
C05324=1029.414,62.079,402.765,168.336,44.651,158.327
C05325=1029.421,62.329,402.747,168.339,44.649,158.327
C05326=1029.428,62.577,402.730,168.340,44.647,158.327
C05327=1029.434,62.827,402.712,168.343,44.645,158.327
C05328=1029.440,63.077,402.696,168.345,44.643,158.327
C05329=1029.447,63.326,402.679,168.348,44.641,158.326
C05330=1029.453,63.576,402.661,168.350,44.639,158.326
C05331=1029.459,63.824,402.644,168.353,44.637,158.326
C05332=1029.465,64.074,402.626,168.355,44.635,158.326
C05333=1029.471,64.323,402.609,168.358,44.633,158.326
C05334=1029.477,64.573,402.591,168.359,44.630,158.326
C05335=1029.484,64.822,402.573,168.362,44.628,158.325
C05336=1029.490,65.071,402.556,168.364,44.626,158.325
C05337=1029.496,65.321,402.538,168.367,44.624,158.325
C05338=1029.502,65.570,402.521,168.369,44.623,158.325
C05339=1029.508,65.819,402.503,168.372,44.620,158.325
C05340=1029.515,66.069,402.486,168.374,44.618,158.325
C05341=1029.521,66.318,402.468,168.376,44.616,158.324
C05342=1029.527,66.568,402.450,168.379,44.614,158.324
C05343=1029.533,66.816,402.434,168.381,44.612,158.324
C05344=1029.539,67.066,402.416,168.383,44.610,158.324
C05345=1029.545,67.315,402.398,168.386,44.608,158.324
C05346=1029.552,67.564,402.380,168.389,44.606,158.324
C05347=1029.558,67.814,402.362,168.391,44.604,158.324
C05348=1029.564,68.062,402.345,168.393,44.602,158.323
C05349=1029.570,68.312,402.327,168.395,44.600,158.323
C05350=1029.576,68.562,402.309,168.398,44.598,158.323
C05351=1029.583,68.811,402.292,168.400,44.596,158.323
C05352=1029.589,69.060,402.274,168.403,44.594,158.323
C05353=1029.594,69.309,402.257,168.405,44.592,158.323
C05354=1029.600,69.559,402.239,168.408,44.590,158.322
C05355=1029.608,69.808,402.221,168.410,44.588,158.322
C05356=1029.613,70.057,402.203,168.412,44.585,158.322
C05357=1029.619,70.307,402.185,168.414,44.583,158.322
C05358=1029.625,70.556,402.167,168.417,44.582,158.322
C05359=1029.632,70.805,402.150,168.420,44.580,158.322
C05360=1029.638,71.054,402.132,168.422,44.578,158.321
C05361=1029.644,71.304,402.114,168.424,44.576,158.321
C05362=1029.650,71.553,402.096,168.426,44.573,158.321
C05363=1029.656,71.803,402.078,168.429,44.571,158.321
C05364=1029.663,72.052,402.060,168.431,44.569,158.321
C05365=1029.669,72.301,402.043,168.434,44.567,158.321
C05366=1029.675,72.550,402.025,168.436,44.566,158.321
C05367=1029.681,72.800,402.007,168.438,44.564,158.320
C05368=1029.687,73.049,401.988,168.441,44.562,158.320
C05369=1029.693,73.298,401.971,168.443,44.559,158.320
C05370=1029.700,73.548,401.953,168.446,44.557,158.320
C05371=1029.705,73.796,401.935,168.448,44.555,158.320
C05372=1029.712,74.046,401.917,168.451,44.553,158.320
C05373=1029.718,74.296,401.899,168.453,44.551,158.319
C05374=1029.724,74.544,401.881,168.455,44.549,158.319
C05375=1029.730,74.793,401.863,168.457,44.547,158.319
C05376=1029.736,75.043,401.845,168.460,44.545,158.319
C05377=1029.743,75.292,401.827,168.462,44.543,158.319
C05378=1029.748,75.541,401.809,168.465,44.541,158.319
C05379=1029.756,75.827,401.789,168.467,44.539,158.318
C05380=1029.763,76.112,401.768,168.470,44.537,158.318
C05381=1029.770,76.397,401.747,168.473,44.534,158.318
C05382=1029.777,76.683,401.727,168.476,44.532,158.318
C05383=1029.784,76.932,401.709,168.478,44.530,158.318
C05384=1029.789,77.181,401.691,168.481,44.527,158.317
C05385=1029.796,77.431,401.672,168.482,44.526,158.317
C05386=1029.802,77.680,401.655,168.485,44.524,158.317
C05387=1029.808,77.929,401.636,168.487,44.522,158.317
C05388=1029.814,78.178,401.618,168.490,44.520,158.317
C05389=1029.820,78.428,401.600,168.493,44.518,158.317
C05390=1029.826,78.677,401.582,168.495,44.516,158.317
C05391=1029.833,78.926,401.563,168.497,44.514,158.316
C05392=1029.838,79.175,401.546,168.499,44.512,158.316
C05393=1029.845,79.425,401.527,168.502,44.510,158.316
C05394=1029.850,79.675,401.508,168.504,44.508,158.316
C05395=1029.856,79.923,401.490,168.507,44.506,158.316
C05396=1029.862,80.173,401.472,168.509,44.504,158.316
C05397=1029.868,80.422,401.453,168.511,44.502,158.315
C05398=1029.875,80.671,401.435,168.514,44.500,158.315
C05399=1029.881,80.921,401.417,168.516,44.498,158.315
C05400=1029.887,81.169,401.399,168.519,44.496,158.315
C05401=1029.893,81.419,401.381,168.521,44.494,158.315
C05402=1029.899,81.668,401.362,168.524,44.492,158.315
C05403=1029.906,81.917,401.343,168.525,44.490,158.314
C05404=1029.911,82.166,401.326,168.528,44.488,158.314
C05405=1029.917,82.416,401.307,168.530,44.486,158.314
C05406=1029.923,82.665,401.289,168.533,44.484,158.314
C05407=1029.929,82.915,401.270,168.536,44.482,158.314
C05408=1029.936,83.164,401.251,168.538,44.480,158.314
C05409=1029.942,83.413,401.233,168.540,44.479,158.314
C05410=1029.948,83.662,401.215,168.542,44.477,158.313
C05411=1029.954,83.911,401.196,168.545,44.474,158.313
C05412=1029.960,84.161,401.179,168.547,44.472,158.313
C05413=1029.967,84.410,401.160,168.550,44.470,158.313
C05414=1029.972,84.659,401.141,168.552,44.468,158.313
C05415=1029.979,84.909,401.123,168.555,44.466,158.313
C05416=1029.984,85.157,401.104,168.557,44.465,158.312
C05417=1029.991,85.406,401.086,168.559,44.463,158.312
C05418=1029.997,85.656,401.068,168.561,44.460,158.312
C05419=1030.003,85.905,401.049,168.564,44.458,158.312
C05420=1030.010,86.154,401.031,168.567,44.456,158.312
C05421=1030.016,86.404,401.012,168.569,44.454,158.312
C05422=1030.022,86.654,400.993,168.572,44.452,158.312
C05423=1030.027,86.902,400.975,168.573,44.451,158.311
C05424=1030.034,87.151,400.956,168.576,44.448,158.311
C05425=1030.040,87.400,400.938,168.578,44.446,158.311
C05426=1030.046,87.650,400.920,168.581,44.444,158.311
C05427=1030.053,87.899,400.901,168.583,44.442,158.311
C05428=1030.059,88.148,400.883,168.586,44.440,158.311
C05429=1030.066,88.397,400.864,168.588,44.438,158.310
C05430=1030.071,88.647,400.845,168.591,44.436,158.310
C05431=1030.077,88.897,400.827,168.593,44.434,158.310
C05432=1030.084,89.146,400.808,168.595,44.432,158.310
C05433=1030.090,89.395,400.789,168.598,44.430,158.310
C05434=1030.096,89.643,400.771,168.600,44.428,158.309
C05435=1030.103,89.892,400.753,168.603,44.426,158.309
C05436=1030.108,90.142,400.733,168.605,44.424,158.309
C05437=1030.114,90.392,400.715,168.608,44.422,158.309
C05438=1030.120,90.641,400.696,168.609,44.420,158.309
C05439=1030.126,90.890,400.677,168.612,44.418,158.309
C05440=1030.132,91.140,400.658,168.615,44.416,158.309
C05441=1030.139,91.389,400.640,168.617,44.414,158.308
C05442=1030.145,91.638,400.621,168.620,44.412,158.308
C05443=1030.152,91.923,400.599,168.622,44.410,158.308
C05444=1030.158,92.208,400.578,168.625,44.408,158.308
C05445=1030.165,92.493,400.556,168.627,44.406,158.308
C05446=1030.173,92.778,400.534,168.631,44.404,158.308
C05447=1030.178,93.027,400.515,168.633,44.402,158.308
C05448=1030.185,93.277,400.496,168.635,44.400,158.307
C05449=1030.191,93.526,400.477,168.637,44.398,158.307
C05450=1030.197,93.775,400.459,168.640,44.396,158.307
C05451=1030.203,94.025,400.439,168.642,44.394,158.307
C05452=1030.209,94.274,400.421,168.645,44.392,158.307
C05453=1030.216,94.523,400.402,168.648,44.390,158.307
C05454=1030.221,94.772,400.383,168.650,44.388,158.306
C05455=1030.228,95.021,400.364,168.652,44.386,158.306
C05456=1030.233,95.271,400.345,168.654,44.384,158.306
C05457=1030.240,95.520,400.326,168.657,44.382,158.306
C05458=1030.245,95.769,400.307,168.660,44.380,158.306
C05459=1030.252,96.019,400.288,168.662,44.378,158.306
C05460=1030.258,96.268,400.270,168.664,44.376,158.305
C05461=1030.264,96.517,400.250,168.667,44.374,158.305
C05462=1030.271,96.766,400.231,168.669,44.372,158.305
C05463=1030.276,97.015,400.212,168.671,44.370,158.305
C05464=1030.283,97.264,400.193,168.674,44.368,158.305
C05465=1030.289,97.514,400.174,168.676,44.366,158.305
